// TwinCAT 3 PLC project DL_Cryo
// ProgramVersion: 3.1.4023.0
// libraries:
//   ESO LDC Comm Common Library, * (ESO)
//   ESO LDC Comm Serial Library, * (ESO)
//   ESO LDC Motor Library, * (ESO)
//   ESO LDC Shutter Library, * (ESO)
//   ESO LDC Timer Library, * (ESO)
//   Tc2_Standard, * (Beckhoff Automation GmbH)
//   Tc2_System, * (Beckhoff Automation GmbH)
//   Tc2_Utilities, * (Beckhoff Automation GmbH)
//   Tc3_Module, * (Beckhoff Automation GmbH)
//   VisuDialogs, * (System)
//   VisuSymbols,3.5.10.0,System
// project tree:
//   / CameraTrigIO.TcTTO, GlobalTextList.TcGTLO, PlcTask.TcTTO
//   DUTs/Enumerator/Devices/ E_JANSSEN_CADM2_FAIL_SAFE_STATE.TcDUT, E_JANSSEN_CMD_TYPE.TcDUT, E_JANSSEN_ERROR.TcDUT, E_JANSSEN_STATUS.TcDUT, E_SA_CH_CMD.TcDUT, E_SA_CH_ERROR.TcDUT, E_SA_POS_ELT_STATE.TcDUT, E_SA_POS_ELT_SUBSTATE.TcDUT, E_SA_POS_SM_STATE.TcDUT, E_SA_RPC_ERROR.TcDUT
//   DUTs/Structures/Comm/ T_JANSSEN_CALIBTATION_VALUES.TcDUT
//   DUTs/Structures/Devices/ T_JANSSEN_CFG.TcDUT, T_JANSSEN_CH_CTRL.TcDUT, T_JANSSEN_COMMAND.TcDUT, T_JANSSEN_CTRL.TcDUT, T_JANSSEN_INFO.TcDUT, T_JANSSEN_READING.TcDUT, T_JANSSEN_STAT.TcDUT, T_SA_CH_STATE.TcDUT, T_SA_DEV_STATUS.TcDUT, T_SCIFY_FILTER_WHEEL_CFG.TcDUT, T_SCIFY_FILTER_WHEEL_STAT.TcDUT
//   GVLs/ GVL_Cryo_Temperatures.TcGVL, GVL_DL_Scanning_Homming.TcGVL
//   POUs/ CameraTrig.TcPOU, FB_Cryostat_State.TcPOU, MAIN.TcPOU
//   POUs/FILTER_WHEEL/ FB_SCIFY_FILTER_WHEEL_FW102C.TcPOU
//   VISUs/ DL_Servo_1_Config.TcVIS, DL_Servo_1_Control.TcVIS, Filter_Wheel.TcVIS, GUI_DL_2.TcVIS, GUI_TIME_INFORMATION.TcVIS, Shutter_1.TcVIS, TipTilt_Servo_1.TcVIS, VisualizationManager.TcVMO (not stored)

CONFIGURATION DL_Cryo
    RESOURCE PLC ON TwinCAT3
        TASK CameraTrigIO(INTERVAL := T#1ms, PRIORITY := 1);
        TASK PlcTask(INTERVAL := T#10ms, PRIORITY := 9);
        PROGRAM CameraTrig WITH CameraTrigIO : CameraTrig;
        PROGRAM MAIN WITH PlcTask : MAIN;
    END_RESOURCE
END_CONFIGURATION

// ---- DUTs/Enumerator/Devices/E_JANSSEN_CADM2_FAIL_SAFE_STATE.TcDUT
{attribute 'qualified_only'}
// 'strict' cannot be used since we mix our own codes with TC codes
//{attribute 'strict'}
TYPE E_JANSSEN_CADM2_FAIL_SAFE_STATE :
(
	OK		 						:= 0,
	UPPER_VOLTAGE_RAIL_IS_MISSING,
	LOWER_VOLTAGE_RAIL_IS_MISSING,	
	THERMAL_OVERLOAD,
	OVER_CURRENT_100US_UPPER_RAIL,
	OVER_CURRENT_1MS_UPPER_RAIL,
	OVER_CURRENT_100US_LOWER_RAIL,
	OVER_CURRENT_1MS_LOWER_RAIL	
);
END_TYPE

// ---- DUTs/Enumerator/Devices/E_JANSSEN_CMD_TYPE.TcDUT
{attribute 'qualified_only'}
{attribute 'strict'}
TYPE E_JANSSEN_CMD_TYPE :
(
	INIT := 0,	// Commands for system initialisation
	READ,		// Commands for Reading status
	CFG,		// Commands for Configuring channels
	CTRL		// Commands for Controlling positioners, e.g. CAL, REF, MOVE, STOP
);
END_TYPE

// ---- DUTs/Enumerator/Devices/E_JANSSEN_ERROR.TcDUT
{attribute 'qualified_only'}
{attribute 'strict'}
TYPE E_JANSSEN_ERROR :
(
	OK				:= 16#0000,
	NOT_IN_OP_STATE	:= 16#0001,
	NOT_INIT		:= 16#0002,
	TIMEOUT			:= 16#0004,
	COMM			:= 16#0008,
	WRONG_STATE		:= 16#0010,
	NOT_IDLE		:= 16#0020
);
END_TYPE

// ---- DUTs/Enumerator/Devices/E_JANSSEN_STATUS.TcDUT
{attribute 'qualified_only'}
{attribute 'strict'}
TYPE E_JANSSEN_STATUS :
(
	NOT_INIT	:= -1,
	IDLE		:= 0,
	ERROR		:= 1,
	BUSY		:= 2
);
END_TYPE

// ---- DUTs/Enumerator/Devices/E_SA_CH_CMD.TcDUT
{attribute 'qualified_only'}
{attribute 'strict'}
TYPE E_SA_CH_CMD :
(
	NONE	:= 0,
	RESET,
	CALIB,
	REF,
	ENABLE,
	DISABLE,
	ENABLE_BASE_DRIVE,
	DISABLE_BASE_DRIVE,
	ENABLE_SERVO_DRIVE,
	DISABLE_SERVO_DRIVE,
	ENABLE_FLEX_DRIVE,
	DISABLE_FLEX_DRIVE,
	STOP,
	MOV,
	MOVE_TO_SETPOINT,
	EMERGENCY_STOP,
	SET_POINT_ACHIEVED
);
END_TYPE

// ---- DUTs/Enumerator/Devices/E_SA_CH_ERROR.TcDUT
{attribute 'qualified_only'}
// 'strict' cannot be used since we mix our own codes with TC codes
//{attribute 'strict'}
TYPE E_SA_CH_ERROR :
(
	OK				:= 0,
	HW_NOT_OP,
	CONFIG,				// Configuration problem, e.g. pointers not set.		
	LOCAL,			
	SETPOS,
	STOP,
	
	ABORT,
	SW_LIMIT_LOWER,
	SW_LIMIT_UPPER,
	ENABLE,
	CTRL,				// MCS2 controller error
	COMM				// MCS2 controller communication problem

);
END_TYPE

// ---- DUTs/Enumerator/Devices/E_SA_POS_ELT_STATE.TcDUT
{attribute 'qualified_only'}
{attribute 'strict'}
TYPE E_SA_POS_ELT_STATE :
(
	NONE	:= 0,
	NOTOP,
	OP
);
END_TYPE

// ---- DUTs/Enumerator/Devices/E_SA_POS_ELT_SUBSTATE.TcDUT
{attribute 'qualified_only'}
{attribute 'strict'}
TYPE E_SA_POS_ELT_SUBSTATE :
(
	NONE					:= 0,
	
	NOTOP_NOTREADY			:= 100,
	NOTOP_READY				:= 101,
	NOTOP_INITIALIZING		:= 102,
	NOTOP_ABORTING			:= 107,
	
	NOTOP_ERROR				:= 199,
	
	
	OP_STANDSTILL			:= 216,            
	OP_MOVING				:= 217,
	OP_SETTING_POS			:= 218,
	OP_STOPPING				:= 219,
	
	OP_ERROR				:= 299
);
END_TYPE

// ---- DUTs/Enumerator/Devices/E_SA_POS_SM_STATE.TcDUT
{attribute 'qualified_only'}
{attribute 'strict'}
TYPE E_SA_POS_SM_STATE :
(
	// Positioner State Machine States
	NOT_READY := 0,	// The system just started.
	CALIB,			// The Positioner is Calibrating
	INIT,			// The Positioner is INITialising/REFerencing
	POST_INIT,		// In POST_INIT we calibrate REF and read CFG once.
	CALIB_REF,		// Calibrate REF position.
	READY,			// NOT OPERATIONAL / READY (i.e. REFerenced)
	
	OP,				// Positioner is Operational
	ERROR,			// Positioner is in error
	
	BASE_DRIVE_MODE, // Janssen controller Basic Drive Mode 
	MOVING,			// Positioner is moving in Basic Drive Mode
	
	STOP,			// Positioner is stopping in Basic Drive Mode OR Exiting a Mode
 	
	
	FLEX_DRIVE_MODE, // Janssen controller external input mode
	
	SERVO_DRIVE_MODE, // ENABLE Janssen controller Servo Drive Mode
	DISABLE_SERVO_DRIVE_MODE, //Disable Janssen controller Servo Drive Mode
	MOVING_TO_SETPOINT,// 3 positioners are Moving to their respective set points in Servo Drive Mode
	EMERGENCY_STOP,    // Emergency stop to halt the positioners
	MOVING_TO_SET_POINT 
	
);
END_TYPE

// ---- DUTs/Enumerator/Devices/E_SA_RPC_ERROR.TcDUT
{attribute 'qualified_only'}
//{attribute 'strict'}
TYPE E_SA_RPC_ERROR :
(
	OK						:= 0,
	NOT_OP					:= -1,			
	NOT_NOTOP_READY			:= -2,			
	NOT_NOTOP_NOTREADY		:= -3,			
	LOCAL					:= -4,			
	SW_LIMIT_LOWER			:= -5,			
	SW_LIMIT_UPPER			:= -6,			
	CHANNEL					:= -7,			
	VEL_ZERO				:= -8,			
	VEL_NEG					:= -9,			
	VEL_MAX					:= -10,			
	CH_NOT_OP				:= -11,
	CTRL_ERROR				:= -12,
	MOVING					:= -13,
	COMM					:= -14	// MCS2 Controller communication problem			
);
END_TYPE

// ---- DUTs/Structures/Comm/T_JANSSEN_CALIBTATION_VALUES.TcDUT
TYPE T_JANSSEN_CALIBTATION_VALUES :
STRUCT
	nGainSetting:				DINT;
	nUpperThresholdValue:		DINT;
	nLowerThresholdValue:		DINT;
END_STRUCT
END_TYPE

// ---- DUTs/Structures/Devices/T_JANSSEN_CFG.TcDUT
TYPE T_JANSSEN_CFG EXTENDS T_RS_BASE_CFG :
STRUCT
	
    //
	// List of Monitoring commands in PRE-OPERATION.
	// Executed before the Positioner has been Referenced/initialised.
	//
	{attribute 'OPC.UA.DA' := '0'}
	cmdList_NOT_READY:	ARRAY [0..15] OF T_JANSSEN_COMMAND := [
							(cmd := 'GFS 1',     	nReplies := 1),
							(cmd := 'GFS 2',     	nReplies := 1),
							(cmd := 'GFS 3',     	nReplies := 1),
							(cmd := 'FBXT', 		nReplies := 1),
							(cmd := 'STP 1', 		nReplies := 1),
							(cmd := 'STP 2', 		nReplies := 1),
							(cmd := 'STP 3', 		nReplies := 1),
							(cmd := '', 			nReplies := 0),
							(cmd := '', 			nReplies := 0)];
	//
	// INIT commands.
	// Executed during Initialisation, before going to OPERATIONAL.
	//
	{attribute 'OPC.UA.DA' := '0'}
	cmdList_Init:	ARRAY [0..7] OF T_JANSSEN_COMMAND := [							
							(cmd := '/GBR USB', 	nReplies := 1),
							(cmd := '', 			nReplies := 0)];

	//
	// List of commands to SET Channel/Positioner Configuration.
	// Note the # and *** characters !!!
	// The actual command will be set like this:
	//    #   will be replaced with channel number
	//    *** will be replaced with a value
	// Example:
	//    ':CHAN#:PCON:OPT ***' => ':CHAN1:PCON:OPT 256'
	//
	// Important NOTE:
	// At this stage RLIM:MIN and RLIM:MAX are disabled, i.e. = 0.
	// The actual limits will be set at the E_SA_POS_SM_STATE.CALIB_REF stage,
	// see M_SetCmdList().
	//
	// These commands are sent only once, just before the positioner is 
	// commanded to Reference (INIT).
	//
	{attribute 'OPC.UA.DA' := '0'}
	cmdList_CfgSet:	ARRAY [0..15] OF T_JANSSEN_COMMAND := [						
							(cmd := '/GBR RS422', 			nReplies := 1),
							(cmd := '/MODLIST', 			nReplies := 1),
							(cmd := 'FBXT', 				nReplies := 1),
							(cmd := 'STP 1', 				nReplies := 1),
							(cmd := 'STP 2', 				nReplies := 1),
							(cmd := 'STP 3', 				nReplies := 1),
							(cmd := 'MLS 4 1', 				nReplies := 1), // Get calibration values
							(cmd := 'MLS 4 2', 				nReplies := 1), // Get calibration values
							(cmd := 'MLS 4 3', 				nReplies := 1), // Get calibration values
							(cmd := 'FBST', 				nReplies := 1), //// Get status position control
							//(cmd := '/VER', 		nReplies := 1),
							//(cmd := 'FBEN CBS10-RLS 300 CBS10-RLS 300 CBS10-RLS 300 1 293', 	nReplies := 1),
							(cmd := '', 					nReplies := 0),			
							//(cmd := ':CHAN#:INP:THR ***', 		nReplies := 0),							
							//(cmd := ':CHAN#:RLIM:MIN 0', 		nReplies := 0),
							(cmd := '', 		nReplies := 0)];
							

	//				
	// List of commands to GET Channel/Positioner Configuration.
	// These commands are sent from the moment the SW started till the positioner 
	// has been Calibrated or Referenced (INIT).
	// Once the Positioer is Ready, these commans are not sent any more.
	//
	{attribute 'OPC.UA.DA' := '0'}
	cmdList_POST_INIT:	ARRAY [0..15] OF T_JANSSEN_COMMAND := [							
							(cmd := '/VER', 		nReplies := 1),
							(cmd := '', 		nReplies := 0)];
							

	

	//
	// List of Monitoring commands in OPERATION.
	// Executed once the Positioner has been Referenced/initialised.
	//
	{attribute 'OPC.UA.DA' := '0'}
	cmdList_Mon:	ARRAY [0..15] OF T_JANSSEN_COMMAND := [
							(cmd := 'GFS 1', 	nReplies := 1),
							(cmd := 'GFS 2', 	nReplies := 1),
							(cmd := 'GFS 3', 	nReplies := 1),
							(cmd := 'FBST', 	nReplies := 1),
							(cmd := 'CGVA 4', 	nReplies := 1),						
							(cmd := '', 		nReplies := 0)];
							
	// Janssen controller flex drive mode
	//Command EXT [ADDR] [DIR] [FREQ] [RSS] [TEMP] [STAGE] [DF]
	cmdList_enable_flex_drive:		ARRAY [0..15] OF T_JANSSEN_COMMAND := [
										(cmd := 'EXT 1 1 600 100 293 CLA2601 1', 	nReplies := 1),						
										(cmd := '', 		nReplies := 0)];
	//Disable flex drive
	//Command FBXT
	//Response (example) Control loop disabled.
	cmdList_disable_flex_drive:	ARRAY [0..15] OF T_JANSSEN_COMMAND := [
										(cmd := 'STP 1', 	nReplies := 1),
										(cmd := 'STP 2', 	nReplies := 1),
										(cmd := 'STP 3', 	nReplies := 1),						
										(cmd := '', 		nReplies := 0)];

	// Janssen controller Servo Drive Mode
	// Command FBEN [STAGE1] [FREQ1] [STAGE2] [FREQ2] [STAGE3] [FREQ3] [DF] [TEMP]		
	cmdList_enable_servo_drive:	ARRAY [0..15] OF T_JANSSEN_COMMAND := [
								(cmd := 'FBEN CBS10-RLS 300 CBS10-RLS 300 CBS10-RLS 300 1 293', 	nReplies := 1),						
								(cmd := '', 		nReplies := 0)];
								
	//Disable servo drive
	//Command FBXT
	//Response (example) Control loop disabled.
	cmdList_disable_servo_drive:	ARRAY [0..15] OF T_JANSSEN_COMMAND := [
								(cmd := 'FBXT', 	nReplies := 1),
								(cmd := 'STP 1', 	nReplies := 1),
								(cmd := 'STP 2', 	nReplies := 1),
								(cmd := 'STP 3', 	nReplies := 1),						
								(cmd := '', 		nReplies := 0)];
	
	// 3 positioners are Moving to their respective set points in Servo Drive Mode
	//Command FBCS [SP1] [ABS] [SP2] [ABS] [SP3] [ABS]
	//Command (example, SP in [m]) FBCS -1e-3 0 1e-3 1 1.23e-4 1
	//Command (example, SP in [rad]) FBCS 6.28 0 0 0 0 0
	//Response (example) Control loop setpoints set.
	
	cmdList_moving_to_setpoint:	ARRAY [0..15] OF T_JANSSEN_COMMAND := [
								(cmd := 'FBCS -1e-3 0 1e-3 1 1.23e-4 1', 	nReplies := 1),						
								(cmd := '', 		nReplies := 0)];
								
	// Emergency stop to halt the positioners
	cmdList_emergency_stop: ARRAY [0..15] OF T_JANSSEN_COMMAND := [
								(cmd := 'FBES', 	nReplies := 1),						
								(cmd := '', 		nReplies := 0)];
								
	// CSZ – Reset current counter value to zero
	//Command CSZ [ADDR] [CH]
	//Command (example) CSZ 4 1
	//Response (example) Position counter set to 0.
	cmdList_reset_counter_to_zero: ARRAY [0..15] OF T_JANSSEN_COMMAND := [
								(cmd := 'CSZ 4 1', 	nReplies := 1),						
								(cmd := '', 		nReplies := 0)];

	//
	// Array of used channels. Set to TRUE for each used channel.
	// 18 channels max. 6 modules [0..5], 3 connections each [CH1, CH2, CH3].
	// channel = (Module x 3) + (CH-1)
	// For example:
	//   First connection (CH1) of first module (Module0): channel = 0 x 3 + (1-1) = 0
	//   Second connection (CH2) of first module (Module0): channel = 0 x 3 + (2-1) = 1
	//   Third connection (CH3) of third module (Module2): channel = 2 x 3 + (3-1) = 8
	//  
	arrUsedCh:	ARRAY [0..17] 	OF BOOL;	

	//
	// Array of used modules. Set to TRUE for each used module.
	// Automatically populated in method M_Configure().
	//
	arrUsedMod:	ARRAY [0..5] 	OF BOOL;	
	
	// Channel configuration structures
//	arrChCfg:	ARRAY [0..17] OF T_SA_CH_CFG;		

(*
	JANSSEN_GET_BR:		STRING(10) := '/GBR RS422';
	JANSSEN_GET_VER:	STRING(8) := '/VER';
	JANSSEN_MODLIST:	STRING(8) := '/MODLIST';
	//CCC_CMD_GET_VERS:	STRING(8) := '>00V??';
	CCC_CMD_GET_VERS:	STRING(8) := '/GBR';
	//CCC_CMD_RESET:		STRING(8) := '>00u??';
	CCC_CMD_RESET:		STRING(8) := '/GBR';
	CCC_CMD_GET_TEMP:	STRING(8) := '>00H??';
	CCC_CMD_GET_FLOW:	STRING(8) := '>00f??';
	//CCC_CMD_GET_STAT:	STRING(8) := '>00o??';
	CCC_CMD_GET_STAT:	STRING(8) := '/GBR';
	CCC_CMD_SET_HOST:	STRING(8) := '>00J??';
	CCC_CMD_SET_THST:	STRING(8) := '>00T??';
	CCC_CMD_SET_TAMB:	STRING(8) := '>00t??';

	(* List of INIT commands *)
	cmdList_Init:	ARRAY [1..4] OF T_JANSSEN_COMMAND := [
							//(cmd := CCC_CMD_RESET, 		nValues := 4),
							//(cmd := CCC_CMD_GET_VERS, 	nValues := 4),
							//(cmd := CCC_CMD_RESET, 		nValues := 0),
							//(cmd := CCC_CMD_GET_VERS, 	nValues := 0),
							//(cmd := JANSSEN_GET_BR, 	nValues := 4),
							//(cmd := '', 				nValues := 0),
							(cmd := '', 				nValues := 0),
							(cmd := '', 				nValues := 0),
							(cmd := '', 				nValues := 0),
							(cmd := '', 				nValues := 0)];


	(*	List of READ commands *)
	cmdList_Read:	ARRAY [1..4] OF T_JANSSEN_COMMAND := [
							//(cmd := CCC_CMD_GET_STAT, 	nValues := 5), (* 5 bytes *)
							//(cmd := CCC_CMD_GET_TEMP, 	nValues := 5), (* 5 words = 10 bytes*)
							//(cmd := CCC_CMD_GET_FLOW, 	nValues := 3), (* 3 words = 6 bytes *)
							//(cmd := JANSSEN_GET_BR, 	nValues := 4),
							(cmd := '/GBR RS422',       nValues := 1),
							(cmd := '/GBR USB', 		nValues := 1),
							(cmd := '', 				nValues := 0),
							(cmd := '', 				nValues := 0)];
		*)
					

END_STRUCT
END_TYPE

// ---- DUTs/Structures/Devices/T_JANSSEN_CH_CTRL.TcDUT
TYPE T_JANSSEN_CH_CTRL :
STRUCT
	//
	// Control structure for a single channel/positioner.
	//
	
	//
	// Active command.
	// Setting nCmd to something other than NONE will
	// trigger execution of commands REF, STOP, MOV.
	//
	nCmd:	E_SA_CH_CMD := E_SA_CH_CMD.NONE;	// Active command
	
	
	// JANSSEN Servo Drive Mode. METIS CFO PSM
	
	// Enable Servodrive
	
	sStage1:	STRING	:= 'CBS10-RLS'; // Mention here the correct stage
	sStage2:	STRING	:= 'CBS10-RLS'; // Mention here the correct stage
	sStage3:	STRING	:= 'CBS10-RLS'; // Mention here the correct stage
	
	// Step Frequency [1 to 600]
	
	nFreq1:		DINT	:= 300; // Step frequency for actuator 1
	nFreq2:		DINT	:= 300; // Step frequency for actuator 2
	nFreq3:		DINT	:= 300; // Step frequency for actuator 3
	
	// Operating Temperturte
	
	nTemp:		DINT; // In Kelvin
	
	// Drive Factor: 
	
	lrDriveFactor:	LREAL := 1.0; // [0.1 to 3.0] In normal operating conditions, set this value to 1 (or 1.0).
	
	// Setpoints
	lrSetPoint1 : LREAL; //Setpoint 1 position in [m]
	lrSetPoint2 : LREAL; //Setpoint 1 position in [m]
	lrSetPoint3 : LREAL; //Setpoint 1 position in [m]
	
	// Set [ABS] to 1 to enable absolute positioning, otherwise set to 0 (zero). 
	// When using COE / OEM2: absolute positioning is relative to count 0 (zero)9 , 
	//whereas relative positioning is relative to the current count value.
	
	bAbsolutePositioning1 : BOOL;
	bAbsolutePositioning2 : BOOL;
	bAbsolutePositioning3 : BOOL;
	
	//SA
	lrPos:	LREAL;		// Position in User Units, i.e. [deg] or [mm]
	lrOff:	LREAL;		// Position offset in User Units, i.e. [deg] or [mm]
	lrVel:	LREAL;		// Velocity in User Units, i.e. [deg/s] or [mm/sec]
	
END_STRUCT
END_TYPE

// ---- DUTs/Structures/Devices/T_JANSSEN_COMMAND.TcDUT
TYPE T_JANSSEN_COMMAND :
STRUCT
	cmd:		STRING := '';	(* Command to send *)
	nReplies:	UINT;   		(* Number of replies, i.e. reply terminators *)
END_STRUCT
END_TYPE

// ---- DUTs/Structures/Devices/T_JANSSEN_CTRL.TcDUT
TYPE T_JANSSEN_CTRL EXTENDS T_RS_BASE_CTRL :
STRUCT
	// Arrays of structures for Configuration and Control commands.
	// Note that only one positioner is handled in each monitoring cycle.
	{attribute 'OPC.UA.DA' := '0'}
	cmdList:			ARRAY [0..15]	OF T_JANSSEN_COMMAND;	// List of up to 16 Commands per channel
	
END_STRUCT
END_TYPE

// ---- DUTs/Structures/Devices/T_JANSSEN_INFO.TcDUT
TYPE T_JANSSEN_INFO :
STRUCT
(*
	Driver Information

	Change LOG:
	1.0	12/02/2014	- Ported from TC2.
	1.1	13/02/2014	- Addition of input parameters for Model and readout period.
	1.2	20/02/2014	- E_CCC_STATUS.ERROR := 1, to match IODev ICD.
					- Disabled OPC UA for comm instance of FB_RS_COMM.
					- Fixed bug in INIT (wrong pointer used)
					- Bytes swapped for Temperatures and Flows.
					- On error, all values set to 9999. Alarm activated.
	1.3 07/11/2014	- Newest version always for References.
					- Remove Tc2_OpcUa library from References.
					- Renamed library to CCC.library (was CCC_TC3.library)
					- Created lib directory.
	1.4 10/02/2016	- On reboot, the device is in NOT INIT (no error!)
					- On INIT start, error is cleared.
	2.0 2016-08-10	- OPC UA notation with TMC Files
	2.1 2017-02-03	- sCmdSuffix and sReplySuffix passed to comm instance.

*)
	sDate:			STRING(16)	:= '2017-02-03';
	sDescription:	STRING(32) 	:= 'Cabinet Cooling Controller';
	sName:			STRING(16)	:= 'FB_CCC';
	sPlatform:		STRING(16)	:= 'CoDeSys';
	sSynopsis:		STRING(48)	:= 'Cabinet Cooling Controller for models 1HE & 4HE';
	nVersionMajor:	DINT		:= 2;
	nVersionMinor:	DINT		:= 1;

END_STRUCT
END_TYPE

// ---- DUTs/Structures/Devices/T_JANSSEN_READING.TcDUT
TYPE T_JANSSEN_READING :
STRUCT
	Value:	LREAL;
END_STRUCT
END_TYPE

// ---- DUTs/Structures/Devices/T_JANSSEN_STAT.TcDUT
TYPE T_JANSSEN_STAT EXTENDS T_RS_BASE_STAT :
STRUCT
	(* STAT *)
	nRetries:			INT := 0;			// Total number of retries in case of communication problems
	
	bPeriodic:			BOOL := FALSE;		(* Flag if device is reading periodically *)

	sReply:				STRING; 			(* Last Reply to predefined commands*)
	
	sRandomtext_1:				STRING;
	sRandomtext_2:				STRING;
	sRandomtext_3:				STRING;
	sRandomtext_4:				STRING;
	sRandomtext_5:				STRING;
	sRandomtext_6:				STRING;
	sRandomtext_7:				STRING;
	sRandomtext_8:				STRING;
	
	sDeviceID:			STRING(48);
	
	(*Baut rate *)
	sBaud_rate_RS422: 			STRING;
	sBaud_rate_USB: 			STRING;
	sFirmware_Version:			STRING;
	sChannel_1_Stop:			STRING;
	sChannel_2_Stop:			STRING;
	sChannel_3_Stop:			STRING;
	
	sFailSafeState_1:			STRING;
	sFailSafeState_2:			STRING;
	sFailSafeState_3:			STRING;
	
	//  
			
	
	// FBST – Get status position control
	sPositionControlStatus:		STRING;
	
	bPositionControl:			BOOL;
	bMovingToSetPoint:			BOOL;
	bInvalidSetPoint_1:			BOOL;
	bInvalidSetPoint_2:			BOOL;
	bInvalidSetPoint_3:			BOOL;
	
	
	nPositionError_1:			DINT;
	nPositionError_2:			DINT;
	nPositionError_3:			DINT;
	
	// MLS Get calibration values
	sCalibrationValues:			STRING;
	
	nCalibrationValues_Cannel_1:	T_JANSSEN_CALIBTATION_VALUES;
	nCalibrationValues_Cannel_2:	T_JANSSEN_CALIBTATION_VALUES;
	nCalibrationValues_Cannel_3:	T_JANSSEN_CALIBTATION_VALUES;
	
	// CGVA 4 counter values of all three channels
	sCounterValues:				STRING;
	
	nCounterValue_Channel_1:		DINT;
	nCounterValue_Channel_2:		DINT;
	nCounterValue_Channel_3:		DINT;
	
	// Command Error
	sCommandError:				STRING;
	
	//Emergency Stop
	bEmergencyStopEnabled:		BOOL;
	
	//FBCS – Go to setpoint -> Control loop setpoints set
	bPositionControlLoop:		BOOL;
	
	//Servo Drive Control
	bServoDrive:				BOOL:= FALSE;
	sServoDriveStatus:			STRING;
	
	//Flex Control
	bFlexDrive:					BOOL;
	
	// /MODLIST Get a list of all installed modules
	
	sInstalledModules:			ARRAY[1..6] OF STRING;
	
	// CGVA – Get current counter value of all channels
	
	nCounterValues:				ARRAY[1..3] OF DINT;
	
	// Get calibration values.  command specific for Basedrive mode of operation
	//Command MLS [ADDR] [CH]
	//Response [GAIN],[UT],[LT]
	
	sCalibValues_1:				STRING;
	sCalibValues_2:				STRING;
	sCalibValues_3:				STRING;

		
	
	
	
	
	(* Status retrieved with command CCC_CMD_GET_STAT *)
	(* decode CSTAT1 byte *)
	bWarn_cabinet_high:			BOOL;
	bWarn_cabinet_no_control:	BOOL;
	bWarn_outlet_high:			BOOL;
	bWarn_inlet_high:			BOOL;
	bWarn_airflow_insufficient:	BOOL;
	bWarn_coolant_insufficient:	BOOL;
	bWarn_door_open:			BOOL;
	bWarn_relay1_warning:		BOOL;
	bWarn_relay2_alarm:			BOOL;

	(* decode CSTAT2 byte *)
	bFault_temp_sensor_ambient:	BOOL;
	bFault_temp_sensor_cabinet:	BOOL;
	bFault_temp_sensor_inlet:	BOOL;
	bFault_temp_sensor_outlet:	BOOL;
	bFault_analog_supply:		BOOL;
	bFault_digital_supply:		BOOL;
	
	(* Temperatures [degC] retrieved with command CCC_CMD_GET_TEMP *)
	lrTemp_outlet:	LREAL;
	lrTemp_inlet:	LREAL;
	lrTemp_cabinet:	LREAL;
	lrTemp_ambient:	LREAL;
	
	(* Flows [l/h] retrieved with command CCC_CMD_GET_FLOW *)
	lrFlow_1:		LREAL;
	lrFlow_2:		LREAL;
	lrFlow_3:		LREAL;
	
	// SmarACT STATs
	
	//bLocal:			BOOL	:= FALSE;	// if TRUE, device operated from PLC GUI 

	//nErrorCode: 	E_SA_CH_ERROR 	:= E_SA_CH_ERROR.OK;	// Error code 
	//nRpcErrorCode: 	E_SA_RPC_ERROR 	:= E_SA_RPC_ERROR.OK;	// RPC Error code

	bCtrlCommProblem:	BOOL;			// SmarAct MCS2 Controller Comm Problem
	//nCtrlErrorCode: E_SM_ERROR;			// SmarAct MCS2 Controller Error code
	nCtrlState:		E_RS_BASE_STATE;	// SmarAct MCS2 Controller State	

	//sErrorText: 	STRING 	:= 'OK'; 			// Error text 
	//sRpcErrorText: 	STRING 	:= 'OK'; 			// RPC Error text 
	//sStatus: 		STRING 	:= 'OK'; 			// Status in textual form, e.g. 'OFF' 
	
	//
	// Standard ELT States and Substates
	//
	//nState:			E_SA_POS_ELT_STATE 		:= E_SA_POS_ELT_STATE.NOTOP;
	//nSubstate:		E_SA_POS_ELT_SUBSTATE	:= E_SA_POS_ELT_SUBSTATE.NOTOP_NOTREADY;
	
	//sState:			STRING	:= 'NOTOP';
	//sSubstate:		STRING	:= 'NOT READY';

	//
	// Positioner State Machine State.
	// Depending on the State, different command sets will be executed.
	//
	nPosState:			E_SA_POS_SM_STATE := E_SA_POS_SM_STATE.NOT_READY;
	nLastPosState:		E_SA_POS_SM_STATE := E_SA_POS_SM_STATE.NOT_READY;
	

	lrPosTarget:		LREAL;			// Target  position in User Units
	lrPosActual:		LREAL;			// Current position in User Units

	//bConfigured:		BOOL;			// Flag if M_Configure has been executed.	
	bError:				BOOL;
	bEnabled:			BOOL;			// Flag if axis is enabled
	//bInitialised:		BOOL;			// Flag if positioner has been initialised/referenced
	bInPosition:		BOOL;			// Flag if axis is In-Position

	//
	// Channel State parameters read from the controller
	// A channel is a Positioner.
	//
	nCH_STATE:				UDINT;			// Positioner State as UDINT
	{attribute 'OPC.UA.DA' := '0'}
	stState:			T_SA_CH_STATE;	// Positioner State structure, from nSTATE
	
	//
	// Device/Channel/Positioner status in user units, i.e. [pm] and [nd].
	// These values are read periodically.
	// Values are normally huge, e.g. pos=18000000000 [nd].
	//
	{attribute 'OPC.UA.DA' := '0'}
	devStatus:			T_SA_DEV_STATUS; 

END_STRUCT
END_TYPE

// ---- DUTs/Structures/Devices/T_SA_CH_STATE.TcDUT
TYPE T_SA_CH_STATE :
STRUCT
	//
	// Channel State
	// Got with the ':CHAN#:STAT?' command
	//
	bBASE_DRIVE_ENABLED:			BOOL;
	bFLEX_DRIVE_ENABLED:			BOOL;
	bSERVO_DRIVE_ENABLED:			BOOL;
	
	bACTIVELY_MOVING:			BOOL;
	bCLOSED_LOOP_ACTIVE:		BOOL;
	bCALIBRATING:				BOOL;
	bREFERENCING:				BOOL;
	bMOVE_DELAYED:				BOOL;
	bSENSOR_PRESENT:			BOOL;
	bIS_CALIBRATED:				BOOL;
	bIS_REFERENCED:				BOOL;
	bEND_STOP_REACHED:			BOOL;
	bRANGE_LIMIT_REACHED:		BOOL;
	bFOLLOWING_LIMIT_REACHED:	BOOL;
	bMOVEMENT_FAILED:			BOOL;
	bIS_STREAMING:				BOOL;
	bPOSITIONER_OVERLOAD:		BOOL;
	
	bOVER_TEMPERATURE:			BOOL;
	
	bREFERENCE_MARK:			BOOL;
	bIS_PHASED:					BOOL;
	bPOSITIONER_FAULT:			BOOL;
	bAMPLIFIER_ENABLED:			BOOL;
	bIN_POSITION:				BOOL;

	bERROR:						BOOL := TRUE;
	bControllerStateError:			BOOL := TRUE;
END_STRUCT
END_TYPE

// ---- DUTs/Structures/Devices/T_SA_DEV_STATUS.TcDUT
//
// Device/Channel/Positioner status in user units, i.e. [pm] and [nd]
//
TYPE T_SA_DEV_STATUS :
STRUCT
	nCAL_OPT:			DINT;			// Calibration option
	nREF_OPT:			DINT;			// Referencing option
	nPCON_OPT:			DINT;			// Positioner Control Options, 256-'in-pos' flag
	nCLIN:				DINT;			// Control Loop Input, 1-SENSOR
	nTUN_BASE_UNIT:		DINT;			// Positioner Base Unit, 2-meter, 3-degree
	nTUN_BASE_RES:		DINT;			// Positioner Base Resolution, 1x10-9 or 1x10-12
	nTUN_MTYP:			DINT;			// Positioner Movement Type, 0-linear, 1-rotation, etc
	nTUN_RTYP:			DINT;			// Positioner Reference Type, 2-SINGLE_CODED
	nINP_THR:			DINT;			// In Position Threshold [DevU]
	nINP_DEL:			DINT;			// In Position Delay [ms]
	nRLIM_MIN:			LINT;			// MIN Limit [DevU]
	nRLIM_MAX:			LINT;			// MAX Limit [DevU]

	lnPosTarget:		LINT;			// Target  position in Positioner Units
	lnPosActual:		LINT;			// Current position in Positioner Units

END_STRUCT
END_TYPE

// ---- DUTs/Structures/Devices/T_SCIFY_FILTER_WHEEL_CFG.TcDUT
TYPE T_SCIFY_FILTER_WHEEL_CFG EXTENDS T_RS_BASE_CFG :
STRUCT
	
    //
	// List of Monitoring commands in PRE-OPERATION.
	// Executed before the Positioner has been Referenced/initialised.
	//
	{attribute 'OPC.UA.DA' := '0'}
	cmdList_NOT_READY:	ARRAY [0..15] OF T_JANSSEN_COMMAND := [
							(cmd := '*idn?',     	nReplies := 1),
							(cmd := 'pos?',     	nReplies := 1),
							(cmd := 'speed?',     	nReplies := 1),
							(cmd := 'sensors?', 		nReplies := 1),
							(cmd := 'baud?', 		nReplies := 1),
							(cmd := '', 			nReplies := 0),
							(cmd := '', 			nReplies := 0)];
	//
	// INIT commands.
	// Executed during Initialisation, before going to OPERATIONAL.
	//
	{attribute 'OPC.UA.DA' := '0'}
	cmdList_Init:	ARRAY [0..7] OF T_JANSSEN_COMMAND := [							
							(cmd := 'pos?',     	nReplies := 1),
							(cmd := '', 			nReplies := 0)];

	//
	// List of commands to SET Channel/Positioner Configuration.
	// Note the # and *** characters !!!
	// The actual command will be set like this:
	//    #   will be replaced with channel number
	//    *** will be replaced with a value
	// Example:
	//    ':CHAN#:PCON:OPT ***' => ':CHAN1:PCON:OPT 256'
	//
	// Important NOTE:
	// At this stage RLIM:MIN and RLIM:MAX are disabled, i.e. = 0.
	// The actual limits will be set at the E_SA_POS_SM_STATE.CALIB_REF stage,
	// see M_SetCmdList().
	//
	// These commands are sent only once, just before the positioner is 
	// commanded to Reference (INIT).
	//
	{attribute 'OPC.UA.DA' := '0'}
	cmdList_CfgSet:	ARRAY [0..15] OF T_JANSSEN_COMMAND := [						
							(cmd := 'pos=5', 	nReplies := 1),
							(cmd := '', 			nReplies := 0)];
							

	//				
	// List of commands to GET Channel/Positioner Configuration.
	// These commands are sent from the moment the SW started till the positioner 
	// has been Calibrated or Referenced (INIT).
	// Once the Positioer is Ready, these commans are not sent any more.
	//
	{attribute 'OPC.UA.DA' := '0'}
	cmdList_POST_INIT:	ARRAY [0..15] OF T_JANSSEN_COMMAND := [							
							(cmd := '/VER', 		nReplies := 1),
							(cmd := '', 		nReplies := 0)];
							

	

	//
	// List of Monitoring commands in OPERATION.
	// Executed once the Positioner has been Referenced/initialised.
	//
	{attribute 'OPC.UA.DA' := '0'}
	cmdList_Mon:	ARRAY [0..15] OF T_JANSSEN_COMMAND := [
							(cmd := '*idn?',     	nReplies := 1),
							(cmd := 'pos?',     	nReplies := 1),
							(cmd := 'speed?',     	nReplies := 1),
							(cmd := 'sensors?', 	nReplies := 1),
							(cmd := 'baud?', 		nReplies := 1),
							(cmd := '', 			nReplies := 0),			
							(cmd := '', 			nReplies := 0)];
							
	// Janssen controller flex drive mode
	//Command EXT [ADDR] [DIR] [FREQ] [RSS] [TEMP] [STAGE] [DF]
	cmdList_enable_flex_drive:		ARRAY [0..15] OF T_JANSSEN_COMMAND := [
										(cmd := 'EXT 1 1 600 100 293 CLA2601 1', 	nReplies := 1),						
										(cmd := '', 		nReplies := 0)];
	//Disable flex drive
	//Command FBXT
	//Response (example) Control loop disabled.
	cmdList_disable_flex_drive:	ARRAY [0..15] OF T_JANSSEN_COMMAND := [
										(cmd := 'STP 1', 	nReplies := 1),
										(cmd := 'STP 2', 	nReplies := 1),
										(cmd := 'STP 3', 	nReplies := 1),						
										(cmd := '', 		nReplies := 0)];

	// Janssen controller Servo Drive Mode
	// Command FBEN [STAGE1] [FREQ1] [STAGE2] [FREQ2] [STAGE3] [FREQ3] [DF] [TEMP]		
	cmdList_enable_servo_drive:	ARRAY [0..15] OF T_JANSSEN_COMMAND := [
								(cmd := 'FBEN CBS10-RLS 300 CBS10-RLS 300 CBS10-RLS 300 1 293', 	nReplies := 1),						
								(cmd := '', 		nReplies := 0)];
								
	//Disable servo drive
	//Command FBXT
	//Response (example) Control loop disabled.
	cmdList_disable_servo_drive:	ARRAY [0..15] OF T_JANSSEN_COMMAND := [
								(cmd := 'FBXT', 	nReplies := 1),
								(cmd := 'STP 1', 	nReplies := 1),
								(cmd := 'STP 2', 	nReplies := 1),
								(cmd := 'STP 3', 	nReplies := 1),						
								(cmd := '', 		nReplies := 0)];
	
	// 3 positioners are Moving to their respective set points in Servo Drive Mode
	//Command FBCS [SP1] [ABS] [SP2] [ABS] [SP3] [ABS]
	//Command (example, SP in [m]) FBCS -1e-3 0 1e-3 1 1.23e-4 1
	//Command (example, SP in [rad]) FBCS 6.28 0 0 0 0 0
	//Response (example) Control loop setpoints set.
	
	cmdList_moving_to_setpoint:	ARRAY [0..15] OF T_JANSSEN_COMMAND := [
								(cmd := 'FBCS -1e-3 0 1e-3 1 1.23e-4 1', 	nReplies := 1),						
								(cmd := '', 		nReplies := 0)];
								
	// Emergency stop to halt the positioners
	cmdList_emergency_stop: ARRAY [0..15] OF T_JANSSEN_COMMAND := [
								(cmd := 'FBES', 	nReplies := 1),						
								(cmd := '', 		nReplies := 0)];
								
	// CSZ – Reset current counter value to zero
	//Command CSZ [ADDR] [CH]
	//Command (example) CSZ 4 1
	//Response (example) Position counter set to 0.
	cmdList_reset_counter_to_zero: ARRAY [0..15] OF T_JANSSEN_COMMAND := [
								(cmd := 'CSZ 4 1', 	nReplies := 1),						
								(cmd := '', 		nReplies := 0)];

	//
	// Array of used channels. Set to TRUE for each used channel.
	// 18 channels max. 6 modules [0..5], 3 connections each [CH1, CH2, CH3].
	// channel = (Module x 3) + (CH-1)
	// For example:
	//   First connection (CH1) of first module (Module0): channel = 0 x 3 + (1-1) = 0
	//   Second connection (CH2) of first module (Module0): channel = 0 x 3 + (2-1) = 1
	//   Third connection (CH3) of third module (Module2): channel = 2 x 3 + (3-1) = 8
	//  
	arrUsedCh:	ARRAY [0..17] 	OF BOOL;	

	//
	// Array of used modules. Set to TRUE for each used module.
	// Automatically populated in method M_Configure().
	//
	arrUsedMod:	ARRAY [0..5] 	OF BOOL;	
	
	// Channel configuration structures
//	arrChCfg:	ARRAY [0..17] OF T_SA_CH_CFG;		

(*
	JANSSEN_GET_BR:		STRING(10) := '/GBR RS422';
	JANSSEN_GET_VER:	STRING(8) := '/VER';
	JANSSEN_MODLIST:	STRING(8) := '/MODLIST';
	//CCC_CMD_GET_VERS:	STRING(8) := '>00V??';
	CCC_CMD_GET_VERS:	STRING(8) := '/GBR';
	//CCC_CMD_RESET:		STRING(8) := '>00u??';
	CCC_CMD_RESET:		STRING(8) := '/GBR';
	CCC_CMD_GET_TEMP:	STRING(8) := '>00H??';
	CCC_CMD_GET_FLOW:	STRING(8) := '>00f??';
	//CCC_CMD_GET_STAT:	STRING(8) := '>00o??';
	CCC_CMD_GET_STAT:	STRING(8) := '/GBR';
	CCC_CMD_SET_HOST:	STRING(8) := '>00J??';
	CCC_CMD_SET_THST:	STRING(8) := '>00T??';
	CCC_CMD_SET_TAMB:	STRING(8) := '>00t??';

	(* List of INIT commands *)
	cmdList_Init:	ARRAY [1..4] OF T_JANSSEN_COMMAND := [
							//(cmd := CCC_CMD_RESET, 		nValues := 4),
							//(cmd := CCC_CMD_GET_VERS, 	nValues := 4),
							//(cmd := CCC_CMD_RESET, 		nValues := 0),
							//(cmd := CCC_CMD_GET_VERS, 	nValues := 0),
							//(cmd := JANSSEN_GET_BR, 	nValues := 4),
							//(cmd := '', 				nValues := 0),
							(cmd := '', 				nValues := 0),
							(cmd := '', 				nValues := 0),
							(cmd := '', 				nValues := 0),
							(cmd := '', 				nValues := 0)];


	(*	List of READ commands *)
	cmdList_Read:	ARRAY [1..4] OF T_JANSSEN_COMMAND := [
							//(cmd := CCC_CMD_GET_STAT, 	nValues := 5), (* 5 bytes *)
							//(cmd := CCC_CMD_GET_TEMP, 	nValues := 5), (* 5 words = 10 bytes*)
							//(cmd := CCC_CMD_GET_FLOW, 	nValues := 3), (* 3 words = 6 bytes *)
							//(cmd := JANSSEN_GET_BR, 	nValues := 4),
							(cmd := '/GBR RS422',       nValues := 1),
							(cmd := '/GBR USB', 		nValues := 1),
							(cmd := '', 				nValues := 0),
							(cmd := '', 				nValues := 0)];
		*)
					

END_STRUCT
END_TYPE

// ---- DUTs/Structures/Devices/T_SCIFY_FILTER_WHEEL_STAT.TcDUT
TYPE T_SCIFY_FILTER_WHEEL_STAT EXTENDS T_RS_BASE_STAT :
STRUCT
	(* STAT *)
	nRetries:			INT := 0;			// Total number of retries in case of communication problems
	
	bPeriodic:			BOOL := FALSE;		(* Flag if device is reading periodically *)

	sReply:				STRING; 			(* Last Reply to predefined commands*)
	
	sRandomtext_1:				STRING;
	sRandomtext_2:				STRING;
	sRandomtext_3:				STRING;
	sRandomtext_4:				STRING;
	sRandomtext_5:				STRING;
	sRandomtext_6:				STRING;
	sRandomtext_7:				STRING;
	sRandomtext_8:				STRING;
	
	
	
	// SCIFY Filter Wheel
	bBaud_rate_RS232: 			BOOL;
	sBaud_rate_RS232: 			STRING;
	
	sDeviceID:					STRING(48);		// Model number and firmware version
	
	sFilterPosition:			STRING;			// Positions 1-6
	nCurrentFilterPosition:			STRING;			
	
	bFilterSensors:				STRING;
	bMoveSpeed:					STRING;
	
	
	
	/////////////
	(*Baut rate *)
	sBaud_rate_RS422: 			STRING;
	sBaud_rate_USB: 			STRING;
	sFirmware_Version:			STRING;
	sChannel_1_Stop:			STRING;
	sChannel_2_Stop:			STRING;
	sChannel_3_Stop:			STRING;
	
	sFailSafeState_1:			STRING;
	sFailSafeState_2:			STRING;
	sFailSafeState_3:			STRING;
	
	//  
			
	
	// FBST – Get status position control
	sPositionControlStatus:		STRING;
	
	bPositionControl:			BOOL;
	bMovingToSetPoint:			BOOL;
	bInvalidSetPoint_1:			BOOL;
	bInvalidSetPoint_2:			BOOL;
	bInvalidSetPoint_3:			BOOL;
	
	
	nPositionError_1:			DINT;
	nPositionError_2:			DINT;
	nPositionError_3:			DINT;
	
	// MLS Get calibration values
	sCalibrationValues:			STRING;
	
	nCalibrationValues_Cannel_1:	T_JANSSEN_CALIBTATION_VALUES;
	nCalibrationValues_Cannel_2:	T_JANSSEN_CALIBTATION_VALUES;
	nCalibrationValues_Cannel_3:	T_JANSSEN_CALIBTATION_VALUES;
	
	// CGVA 4 counter values of all three channels
	sCounterValues:				STRING;
	
	nCounterValue_Channel_1:		DINT;
	nCounterValue_Channel_2:		DINT;
	nCounterValue_Channel_3:		DINT;
	
	// Command Error
	sCommandError:				STRING;
	
	//Emergency Stop
	bEmergencyStopEnabled:		BOOL;
	
	//FBCS – Go to setpoint -> Control loop setpoints set
	bPositionControlLoop:		BOOL;
	
	//Servo Drive Control
	bServoDrive:				BOOL:= FALSE;
	sServoDriveStatus:			STRING;
	
	//Flex Control
	bFlexDrive:					BOOL;
	
	// /MODLIST Get a list of all installed modules
	
	sInstalledModules:			ARRAY[1..6] OF STRING;
	
	// CGVA – Get current counter value of all channels
	
	nCounterValues:				ARRAY[1..3] OF DINT;
	
	// Get calibration values.  command specific for Basedrive mode of operation
	//Command MLS [ADDR] [CH]
	//Response [GAIN],[UT],[LT]
	
	sCalibValues_1:				STRING;
	sCalibValues_2:				STRING;
	sCalibValues_3:				STRING;

		
	
	
	
	
	(* Status retrieved with command CCC_CMD_GET_STAT *)
	(* decode CSTAT1 byte *)
	bWarn_cabinet_high:			BOOL;
	bWarn_cabinet_no_control:	BOOL;
	bWarn_outlet_high:			BOOL;
	bWarn_inlet_high:			BOOL;
	bWarn_airflow_insufficient:	BOOL;
	bWarn_coolant_insufficient:	BOOL;
	bWarn_door_open:			BOOL;
	bWarn_relay1_warning:		BOOL;
	bWarn_relay2_alarm:			BOOL;

	(* decode CSTAT2 byte *)
	bFault_temp_sensor_ambient:	BOOL;
	bFault_temp_sensor_cabinet:	BOOL;
	bFault_temp_sensor_inlet:	BOOL;
	bFault_temp_sensor_outlet:	BOOL;
	bFault_analog_supply:		BOOL;
	bFault_digital_supply:		BOOL;
	
	(* Temperatures [degC] retrieved with command CCC_CMD_GET_TEMP *)
	lrTemp_outlet:	LREAL;
	lrTemp_inlet:	LREAL;
	lrTemp_cabinet:	LREAL;
	lrTemp_ambient:	LREAL;
	
	(* Flows [l/h] retrieved with command CCC_CMD_GET_FLOW *)
	lrFlow_1:		LREAL;
	lrFlow_2:		LREAL;
	lrFlow_3:		LREAL;
	
	// SmarACT STATs
	
	//bLocal:			BOOL	:= FALSE;	// if TRUE, device operated from PLC GUI 

	//nErrorCode: 	E_SA_CH_ERROR 	:= E_SA_CH_ERROR.OK;	// Error code 
	//nRpcErrorCode: 	E_SA_RPC_ERROR 	:= E_SA_RPC_ERROR.OK;	// RPC Error code

	bCtrlCommProblem:	BOOL;			// SmarAct MCS2 Controller Comm Problem
	//nCtrlErrorCode: E_SM_ERROR;			// SmarAct MCS2 Controller Error code
	nCtrlState:		E_RS_BASE_STATE;	// SmarAct MCS2 Controller State	

	//sErrorText: 	STRING 	:= 'OK'; 			// Error text 
	//sRpcErrorText: 	STRING 	:= 'OK'; 			// RPC Error text 
	//sStatus: 		STRING 	:= 'OK'; 			// Status in textual form, e.g. 'OFF' 
	
	//
	// Standard ELT States and Substates
	//
	//nState:			E_SA_POS_ELT_STATE 		:= E_SA_POS_ELT_STATE.NOTOP;
	//nSubstate:		E_SA_POS_ELT_SUBSTATE	:= E_SA_POS_ELT_SUBSTATE.NOTOP_NOTREADY;
	
	//sState:			STRING	:= 'NOTOP';
	//sSubstate:		STRING	:= 'NOT READY';

	//
	// Positioner State Machine State.
	// Depending on the State, different command sets will be executed.
	//
	nPosState:			E_SA_POS_SM_STATE := E_SA_POS_SM_STATE.NOT_READY;
	nLastPosState:		E_SA_POS_SM_STATE := E_SA_POS_SM_STATE.NOT_READY;
	

	lrPosTarget:		LREAL;			// Target  position in User Units
	lrPosActual:		LREAL;			// Current position in User Units

	//bConfigured:		BOOL;			// Flag if M_Configure has been executed.	
	bError:				BOOL;
	bEnabled:			BOOL;			// Flag if axis is enabled
	//bInitialised:		BOOL;			// Flag if positioner has been initialised/referenced
	bInPosition:		BOOL;			// Flag if axis is In-Position

	//
	// Channel State parameters read from the controller
	// A channel is a Positioner.
	//
	nCH_STATE:				UDINT;			// Positioner State as UDINT
	{attribute 'OPC.UA.DA' := '0'}
	stState:			T_SA_CH_STATE;	// Positioner State structure, from nSTATE
	
	//
	// Device/Channel/Positioner status in user units, i.e. [pm] and [nd].
	// These values are read periodically.
	// Values are normally huge, e.g. pos=18000000000 [nd].
	//
	{attribute 'OPC.UA.DA' := '0'}
	devStatus:			T_SA_DEV_STATUS; 

END_STRUCT
END_TYPE

// ---- GVLs/GVL_Cryo_Temperatures.TcGVL
{attribute 'qualified_only'}
VAR_GLOBAL
	
// Temperature Sensors
	{attribute 'OPC.UA.DA' := '1'}
	Temp_1 : REAL;
	
	{attribute 'OPC.UA.DA' := '1'}
	Temp_2 : REAL;

	{attribute 'OPC.UA.DA' := '1'}
	Temp_3 : REAL;

	{attribute 'OPC.UA.DA' := '1'}
	Temp_4 : REAL;	
	
// Heater 

	{attribute 'OPC.UA.DA' := '1'}
	CryoHeater_1 : UINT;
	
	{attribute 'OPC.UA.DA' := '1'}
	CryoHeater_2 : UINT;
	
	{attribute 'OPC.UA.DA' := '1'}
	CryoHeater_3 : UINT;
END_VAR

// ---- GVLs/GVL_DL_Scanning_Homming.TcGVL
{attribute 'qualified_only'}
VAR_GLOBAL
	{attribute 'OPC.UA.DA':='1'}
	bHomming :BOOL;
	
	{attribute 'OPC.UA.DA':='1'}
	sHommingStatus :STRING;
	
	{attribute 'OPC.UA.DA':='1'}
	bTrigCameraImages :BOOL;
END_VAR

// ---- POUs/CameraTrig.TcPOU
PROGRAM CameraTrig
VAR
bCameraIN_1 AT %I* : BOOL;

bCameraIN_2 AT %I* : BOOL;

bCameraOUT_1 AT %Q* : BOOL;

bCameraOUT_2 AT %Q* : BOOL;

{attribute 'OPC.UA.DA':='1'}
b_Camera_in_1 :BOOL;
{attribute 'OPC.UA.DA':='1'}
b_Camera_in_2 :BOOL;
{attribute 'OPC.UA.DA':='1'}
b_Camera_out_1 :BOOL;
{attribute 'OPC.UA.DA':='1'}
b_Camera_out_2 :BOOL;
END_VAR

b_Camera_in_1 :=   bCameraIN_1; 

b_Camera_in_2 :=   bCameraIN_2; 

 bCameraOUT_1 :=  b_Camera_out_1;

 bCameraOUT_2 :=  b_Camera_out_2;

END_PROGRAM

// ---- POUs/MAIN.TcPOU
PROGRAM MAIN
VAR



// DL Servo
	
{attribute 'OPC.UA.DA':='1'}

DL_Servo_1: FB_MOTOR;

// DL Newport stepper
	
{attribute 'OPC.UA.DA':='1'}
DL_2: FB_MOTOR;

// Camera triggers

//bCameraIN_1 AT %I* : BOOL;

//bCameraIN_2 AT %I* : BOOL;

//bCameraOUT_1 AT %Q* : BOOL;

//bCameraOUT_2 AT %Q* : BOOL;

//{attribute 'OPC.UA.DA':='1'}
//b_Camera_in_1 :BOOL;
//{attribute 'OPC.UA.DA':='1'}
//b_Camera_in_2 :BOOL;
//{attribute 'OPC.UA.DA':='1'}
//b_Camera_out_1 :BOOL;
//{attribute 'OPC.UA.DA':='1'}
//b_Camera_out_2 :BOOL;

{attribute 'OPC.UA.DA':='1'}
fbCryoState : FB_Cryostat_State;

// Homming
iLocalCOntrolStatus : INT;


//Fring Scanning

// Time Stamp
fbGetSystemTime  : GETSYSTEMTIME;
fileTime         : T_FILETIME;
{attribute 'OPC.UA.DA':='1'}
sTime            : STRING;

// NPT PTP

time_info:	FB_TIME;

///

// Filter Wheel

FILTER_WHEEL	:	FB_SCIFY_FILTER_WHEEL_FW102C;

// Accelerometer

in_nVib_X AT %I* :DINT;	
in_nVib_Y AT %I* :DINT;
in_nVib_Z AT %I* :DINT;

{attribute 'OPC.UA.DA':='1'}
nVib_X:	DINT;
{attribute 'OPC.UA.DA':='1'}
nVib_Y:	DINT;
{attribute 'OPC.UA.DA':='1'}
nVib_Z:	DINT;

////
//Shutters
//////
{attribute 'OPC.UA.DA':='1'}
shutter_1:		FB_SHUTTER;


/// Tip-tilt motors
{attribute 'OPC.UA.DA':='1'}
tiptilt_1: FB_MOTOR;




END_VAR


fbCryoState();

DL_Servo_1(sName:='DL_Servo_1', nNOVRAM_DevId:=5, nNOVRAM_Offset:= 1000);

DL_2(sName:='DL_2_Newport', nNOVRAM_DevId:=5, nNOVRAM_Offset:= 2000);

//bCameraOUT_1 := GVL_DL_Scanning_Homming.bTrigCameraImages;


// Time Stamps

fbGetSystemTime(timeLoDW=>fileTime.dwLowDateTime, timeHiDW=>fileTime.dwHighDateTime );
sTime := SYSTEMTIME_TO_STRING( FILETIME_TO_SYSTEMTIME( fileTime ) );

time_info();

// Filter Wheel

FILTER_WHEEL(in_bSimulation:= FALSE, in_sName:= 'FILTER_WHEEL', in_nPeriod:= 1200);

// Vibration from Accelero sensor

nVib_X := in_nVib_X;
nVib_Y := in_nVib_Y;
nVib_Z := in_nVib_Z;

////  Shutters

shutter_1(
	in_sName:= 'Shutter_1', 
	in_bActiveLowClosed:= , 
	in_bActiveLowFault:= , 
	in_bActiveLowOpen:= TRUE, 
	in_bActiveLowSwitch:= , 
	in_bIgnoreClosed:= , 
	in_bIgnoreFault:= , 
	in_bIgnoreOpen:= , 
	in_bInitialState:= , 
	in_nTimeout:= , 
	in_bLogExtTime:= , 
	in_bLog:= );
	
/// Tip-tilt motors

tiptilt_1(sName:='Tip-Tilt_1', nNOVRAM_DevId:=5, nNOVRAM_Offset:= 4000);


//b_Camera_in_1 :=   bCameraIN_1; 

//b_Camera_in_2 :=   bCameraIN_2; 

//b_Camera_out_1 :=  bCameraOUT_1;

//b_Camera_out_2 :=  bCameraOUT_2;

END_PROGRAM

// ---- POUs/FB_Cryostat_State.TcPOU
FUNCTION_BLOCK FB_Cryostat_State
VAR_INPUT
END_VAR
VAR_OUTPUT
END_VAR
VAR
	nCryotemp_1 AT %I* : INT;
	nCryotemp_2 AT %I* : INT;
	nCryotemp_3 AT %I* : INT;
	nCryotemp_4 AT %I* : INT;
	
	nCryoHeater_1 AT %Q* : UINT;
	nCryoHeater_2 AT %Q* : UINT;
	nCryoHeater_3 AT %Q* : UINT;
END_VAR

GVL_Cryo_Temperatures.Temp_1 := nCryotemp_1 /10;

GVL_Cryo_Temperatures.Temp_2 := nCryotemp_2 /10;

GVL_Cryo_Temperatures.Temp_3 := nCryotemp_3 /10;

GVL_Cryo_Temperatures.Temp_4 := nCryotemp_4 /10;

nCryoHeater_1 := GVL_Cryo_Temperatures.CryoHeater_1;
nCryoHeater_1 := GVL_Cryo_Temperatures.CryoHeater_2;
nCryoHeater_1 := GVL_Cryo_Temperatures.CryoHeater_3;

END_FUNCTION_BLOCK

// ---- POUs/FILTER_WHEEL/FB_SCIFY_FILTER_WHEEL_FW102C.TcPOU
FUNCTION_BLOCK FB_SCIFY_FILTER_WHEEL_FW102C EXTENDS FB_RS_BASE
VAR_INPUT
	{attribute 'OPC.UA.DA' := '0'}
	in_nPeriod:	DINT := 10000;	// Interval for periodic reading [ms], default 10000 ms = 10 sec 
END_VAR
VAR_OUTPUT
END_VAR
VAR CONSTANT
	{attribute 'OPC.UA.DA' := '0'}
	//sCmdSuffix:		STRING(16) := '$0D$0A'; // CR LF
	sCmdSuffix:		STRING(16) := '$0D';		// CR
	{attribute 'OPC.UA.DA' := '0'}
	sReplySuffix:	STRING(16) := '$3E';		// >
END_VAR
VAR
	{attribute 'OPC.UA.DA' := '1'}
	cfg:		T_SCIFY_FILTER_WHEEL_CFG;		//  Config parameters
	{attribute 'OPC.UA.DA' := '1'}
	ctrl:		T_JANSSEN_CTRL;					//  Control parameters
	{attribute 'OPC.UA.DA' := '1'}
	{attribute 'OPC.UA.DA.Access' := '1'}
	info:		T_JANSSEN_INFO; 				//  Info parameters - ReadOnly
	{attribute 'OPC.UA.DA' := '1'}
	{attribute 'OPC.UA.DA.Access' := '1'}
	stat:		T_SCIFY_FILTER_WHEEL_STAT;					//  Status parameters - ReadOnly
	{attribute 'OPC.UA.DA' := '1'}
	ch_ctrl:	T_JANSSEN_CH_CTRL;				//  Channel control

	{attribute 'OPC.UA.DA' := '0'}
	comm:		FB_RS_COMM_NO_SIM;					// Instance of generic comm object. OPC UA Disabled!!!
	
	//{attribute 'OPC.UA.DA' := '0'}
	//comm:		FB_RS_COMM_LAKESHORE;	// Instance of Lakeshore customized comm 
	
	(* Pointers *)
	{attribute 'OPC.UA.DA' := '0'}
	ptrCommCfg:		POINTER TO T_RS_COMM_CFG 	:= ADR(comm.cfg);	(* Pointer to comm.cfg instance *)
	{attribute 'OPC.UA.DA' := '0'}
	ptrCommCtrl:	POINTER TO T_RS_COMM_CTRL 	:= ADR(comm.ctrl);	(* Pointer to comm.ctrl instance *)
	{attribute 'OPC.UA.DA' := '0'}
	ptrCommStat:	POINTER TO T_RS_COMM_STAT 	:= ADR(comm.stat);	(* Pointer to comm.stat instance *)
	{attribute 'OPC.UA.DA' := '0'}
	ptrInitCmds:	POINTER TO ARRAY [1..4] OF T_JANSSEN_COMMAND;		(* Pointer to INIT commands *)
	{attribute 'OPC.UA.DA' := '0'}
	ptrReadCmds:	POINTER TO ARRAY [1..4] OF T_JANSSEN_COMMAND;		(* Pointer to READ commands *)


	(* Timers *)
	{attribute 'OPC.UA.DA' := '0'}
	fbTimer:			TON; (* General Timeout *)
	
	(* Misc internal vars *)
	{attribute 'OPC.UA.DA' := '0'}
	cmdCounter:			INT := 1;

END_VAR

// Set references
cfgRef	REF=cfg;
ctrlRef	REF=ctrl;
statRef	REF=stat;


(* Execute comm instance *)
comm(in_sCmdSuffix:=sCmdSuffix, in_sReplySuffix:=sReplySuffix, in_nTimeout:=3000);



// Execute the base class object FB_RS_BASE
SUPER^();

METHOD ActivityInitializing
VAR_INPUT
	bExecute:	BOOL;
END_VAR
VAR_INST
	{attribute 'OPC.UA.DA' := '0'}
    nMethodState:	INT := 0;	// State Machine current state
END_VAR

// SmarACT
SetAction('ActivityInitializing');


IF NOT bExecute THEN
	nMethodState	:= 0;	// Reset the state machine
	cmdCounter		:= -1;	// First init command. CASE 15: will increment it to 0
	//cmdCounter		:= 1;	
	RETURN;
END_IF

// Handle State Machine
CASE nMethodState OF
	0:	// Initialize COMM port
		(* Reset the port *)
		ptrCommCtrl^.nCommand	:= E_RS_COMM_CMD.INIT;
		ptrCommCtrl^.bExecute	:= TRUE;

		(* Start the timer by going false/true *)
		fbTimer (IN := FALSE); (* Reset timer *)
		fbTimer (IN := TRUE, PT := T#5S); (* 5 sec timeout for reply *)

		nMethodState 	:= 15;	// On next cycle wait until the comm port is reset, i.e. idle
		
	15:	// Wait IDLE
		fbTimer (IN := TRUE);
		IF M_GetCommStatus() = E_RS_COMM_STATUS.IDLE  AND M_GetCommInitialised() THEN
			// Communication is IDLE 
			fbTimer (IN := FALSE);	// disable timer 
			stat.sReply		:= ptrCommStat^.sReply;	// Save the reply

			// Extract values from the reply to a stat variable.
			IF ptrCommCtrl^.bHasReply	THEN
				// Index is not important for INIT commands because they don't
				// refer to MODule or CHANnel.
				// We put zero for the input parameter.
				M_ReadReply();	// Index is not important for INIT commands.
			END_IF

			cmdCounter		:= cmdCounter + 1;	// Increment init command index
			fbTimer (IN := FALSE);	// disable timer 
			fbTimer (IN := TRUE, PT := cfg.tDelay_Init); // Wait INIT delay
			bCommProblem	:= FALSE;
			nMethodState 	:= 18;	// Execute next device INIT command
		ELSIF M_GetCommStatus() = E_RS_COMM_STATUS.ERROR  AND fbTimer.ET > T#4900MS THEN
			fbTimer (IN := FALSE);
			SetStatus(E_LAKESHORE_ERROR.COMM, 'ERROR: Communication error');	
			bCommProblem	:= TRUE;
			nEvent := E_SM_EVENT.ERRINIT;
			RETURN;
		ELSIF fbTimer.Q THEN
			// Timer expired after 5 sec. This is an error.
			fbTimer (IN := FALSE);
			SetStatus(E_LAKESHORE_ERROR.TIMEOUT, 'ERROR: Communication timeout');	
			bCommProblem	:= TRUE;
			nEvent := E_SM_EVENT.ERRINIT;
			RETURN;
		END_IF

	
	
	18:	// Wait INIT Delay
		fbTimer (IN := TRUE);
		IF fbTimer.Q THEN
			// Timer expired after 5 sec. This is an error.
			fbTimer (IN := FALSE);
			nMethodState 	:= 20;	// Execute next device INIT command
			RETURN;
		END_IF

	
	
	20:	// INIT DEV
		IF cfg.cmdList_Init[cmdCounter].cmd = '' THEN
			// Device INIT is done. Go to IDLE 
			stat.bInitialised 	:= TRUE;
			cmdCounter			:= 1;
			SetStatus(E_SM_ERROR.OK, 'IDLE');
			nEvent 		:= E_SM_EVENT.INITDONE;
			RETURN;
		END_IF
		
		(* Send INIT command with index cmdCounter *)
		ptrCommCtrl^.nCommand		:= E_RS_COMM_CMD.SEND;
		ptrCommCtrl^.sCmd			:= cfg.cmdList_Init[cmdCounter].cmd;
		ptrCommCtrl^.nNumReplies	:= cfg.cmdList_Init[cmdCounter].nReplies;
		ptrCommCtrl^.bHasReply		:= cfg.cmdList_Init[cmdCounter].nReplies > 0;
		ptrCommCtrl^.bExecute		:= TRUE;
	
		(* Start the timer by going false/true *)
		fbTimer (IN := FALSE); (* Reset timer *)
		fbTimer (IN := TRUE, PT := T#5S); (* 5 sec timeout for reply *)

		// On next cycle wait until the comm port is idle
		nMethodState 	:= 15;	// On next cycle wait until the comm port is idle
	
END_CASE

(*
// Lakeshore
SetAction('ActivityInitializing');


IF NOT bExecute THEN
	nMethodState	:= 0;	// Reset the state machine
	cmdCounter		:= 1;	// Init will start from the first init command
	RETURN;
END_IF

// Handle State Machine
CASE nMethodState OF
	0:	// Set communication parameters and Model configuration

		(* Set comm suffixes for commands and replies *)
		ptrCommCfg^.sCmdSuffix		:= sCmdSuffix;
		ptrCommCfg^.sReplySuffix	:= sReplySuffix;

		// Set monitoring period (input parameter)
		cfg.tDelay_Periodic	:= DINT_TO_TIME(in_nPeriod);
		// Auto monitor, i.e. monitor in Standby_Ready as well
		cfg.bAutoMonitor	:= TRUE; 
		//cfg.bAutoMonitor	:= FALSE;

		(* Set pointer to INIT and READ commands *)
		ptrInitCmds := ADR(cfg.cmdList_Init);
		//ptrReadCmds := ADR(cfg.cmdList_Read);
		ptrReadCmds := ADR(cfg.cmdList_Mon);
		(* Set initial state and status *)
		stat.bInitialised	:= FALSE;
		stat.sReply			:= '';
		stat.sDeviceID		:= '';

		SetStatus(E_SM_ERROR.OK, 'BUSY');

		nMethodState := 10;				// Go to next state, i.e. INIT_COMM

	10:	// Initialize COMM port
		(* Reset the serial port *)
		ptrCommCtrl^.nCommand	:= E_RS_COMM_CMD.INIT;
		ptrCommCtrl^.bExecute	:= TRUE;

		// Init dev will start from the first init command.
		// We set counter to 0. It will be incremented in Wait IDLE.
		cmdCounter	:= 0;

		(* Start the timer by going false/true *)
		fbTimer (IN := FALSE); (* Reset timer *)
		fbTimer (IN := TRUE, PT := T#5S); (* 5 sec timeout for reply *)

		nMethodState 	:= 15;	// On next cycle wait until the comm port is reset, i.e. idle
		
	15:	// Wait IDLE
		fbTimer (IN := TRUE);
		IF comm.stat.nStatus = E_RS_COMM_STATUS.IDLE THEN
			// Communication is IDLE 
			fbTimer (IN := FALSE);	// disable timer 
			 stat.sReply		:= ptrCommStat^.sReply;	// Save the reply
			(*
			IF cmdCounter >= 1 THEN
				// We are IDLE after an INIT command, i.e. CCC_CMD_RESET or CCC_CMD_GET_VERS
				IF ptrInitCmds^ [cmdCounter].cmd = cfg.CCC_CMD_RESET  THEN
					(* No action. Just check proper reply. *)
					IF FIND (stat.sReply, 'N')= 1 THEN
						SetStatus(E_CCC_ERROR.COMM, 'ERROR: Failed to RESET device');
						bCommProblem	:= TRUE;
						nEvent := E_SM_EVENT.ERRINIT;
						RETURN;
					END_IF
				ELSIF ptrInitCmds^ [cmdCounter].cmd = cfg.CCC_CMD_GET_VERS  THEN
					(* Save the reply into stat.sDeviceID. *)
					IF FIND (stat.sReply, 'N')= 1 THEN
						SetStatus(E_CCC_ERROR.COMM, 'ERROR: Command GET_VERS failed');
						bCommProblem	:= TRUE;
						nEvent := E_SM_EVENT.ERRINIT;
						RETURN;
					ELSIF FIND (stat.sReply, 'ESO')<> 2 THEN
						SetStatus(E_CCC_ERROR.COMM, 'ERROR: Failed to get device ID');
						bCommProblem	:= TRUE;
						nEvent := E_SM_EVENT.ERRINIT;
						RETURN;
					ELSE
						stat.sDeviceID	:= MID (stat.sReply, LEN(stat.sReply)-5, 2);
					END_IF
				END_IF
			END_IF
			*)
			// Restart the timer for delay between INIT commands
			fbTimer (IN := FALSE);	// disable timer 
			
			fbTimer (IN := TRUE, PT := cfg.tDelay_Init); // Wait INIT delay
			
			cmdCounter		:= cmdCounter + 1;	// Increment init command index
			bCommProblem	:= FALSE;
			nMethodState 	:= 18;	// Execute next device INIT command
		ELSIF comm.stat.nStatus = E_RS_COMM_STATUS.ERROR THEN
			fbTimer (IN := FALSE);
			SetStatus(E_CCC_ERROR.COMM, 'ERROR: Communication error');	
			bCommProblem	:= TRUE;
			nEvent := E_SM_EVENT.ERRINIT;
			RETURN;
		ELSIF fbTimer.Q THEN
			// Timer expired after 5 sec. This is an error.
			fbTimer (IN := FALSE);
			SetStatus(E_JANSSEN_ERROR.TIMEOUT, 'ERROR: Communication timeout');	
			bCommProblem	:= TRUE;
			nEvent := E_SM_EVENT.ERRINIT;
			RETURN;
		END_IF 

	
	
	18:	// Wait INIT Delay
		fbTimer (IN := TRUE);
		IF fbTimer.Q THEN
			// Timer expired after 5 sec. This is an error.
			fbTimer (IN := FALSE);
			nMethodState 	:= 20;	// Execute next device INIT command
			RETURN;
		END_IF

	
	
	20:	// INIT DEV
		IF ptrInitCmds^ [cmdCounter].cmd = '' THEN
			// Device INIT is done. Go to IDLE 
			stat.bInitialised 	:= TRUE;
			cmdCounter			:= 1;
			SetStatus(E_JANSSEN_STATUS.IDLE, 'IDLE');
			nEvent 		:= E_SM_EVENT.INITDONE;
			RETURN;
		END_IF
		
		
		
		(* Send INIT command with index cmdCounter *)
		ptrCommCtrl^.nCommand		:= E_RS_COMM_CMD.SEND;
		ptrCommCtrl^.sCmd			:= ptrInitCmds^ [cmdCounter].cmd;
		ptrCommCtrl^.nNumReplies	:= 1;
		ptrCommCtrl^.bHasReply		:= TRUE;
		ptrCommCtrl^.bExecute		:= TRUE;
	
		(* Start the timer by going false/true *)
		fbTimer (IN := FALSE); (* Reset timer *)
		fbTimer (IN := TRUE, PT := T#5S); (* 5 sec timeout for reply *)
		
		// On next cycle wait until the comm port is idle
		nMethodState 	:= 15;	// On next cycle wait until the comm port is idle
	
END_CASE
*)
END_METHOD

METHOD ActivityMonitoring
VAR_INPUT
	bExecute:	BOOL;
END_VAR
VAR_INST
	{attribute 'OPC.UA.DA' := '0'}
    nMethodState:	INT := 0;	// State Machine current state
	{attribute 'OPC.UA.DA' := '0'}
	nRetries:		INT := 0;	// Number of retries in case of communication problems
	
	{attribute 'OPC.UA.DA' := '0'}
	nCmdType:		E_JANSSEN_CMD_TYPE := E_JANSSEN_CMD_TYPE.READ;
	{attribute 'OPC.UA.DA' := '0'}
	devCmd:			T_JANSSEN_COMMAND;	// Device command to be sent
	
	{attribute 'OPC.UA.DA' := '0'}
	nCmdIdx:		UINT := 0;	// Command index in specific command list. [0..15]

END_VAR
VAR
	bError:			BOOL;
	
END_VAR

//SmarACT
//
// At least one module must be used.
// If not, don't do anything.
//
(*
IF stat.nNumMod = 0	THEN
	SetAction('ERROR: No Module Used !!!'); 
	SetStatus(E_SM_ERROR.INIT_FAILURE, 'ERROR: No Module Used !!!');
	RETURN;
END_IF
*)
IF NOT cfg.bAutoMonitor AND stat.nSubstate = E_RS_BASE_SUBSTATE.NOTOP_READY THEN
	SetAction('No Monitoring'); 
	SetStatus(E_SM_ERROR.OK, 'IDLE');
	nMethodState	:= 0;	// Reset the state machine
	RETURN;
END_IF

IF NOT bExecute THEN
	SetAction('ActivityMonitoring'); 
	SetStatus(E_SM_ERROR.OK, 'BUSY');
	nMethodState	:= 0;	// Reset the state machine
	nCmdType		:= E_JANSSEN_CMD_TYPE.READ;	// We start with READ commands.
	RETURN;
END_IF

// Handle State Machine
CASE nMethodState OF
	0:	// Get valid channel.
		// This call will check if the current channel is used.
		// If not, it will take next available channel.
		
		//nChIdx	:= M_GetValidChannel(nChIdx);
		
		
		
		// If this is the very first command for the channel,
		// Set commands.
		IF nCmdIdx = 0	THEN
			M_SetCmdList();
		END_IF
		
		
		// Get next command to execute.
		// The command depends on the state of the positioner and 
		// the current index (nCmdIdx) of the command in the list.
		//
		//devCmd	:= M_GetCommand(nCmdIdx);
		devCmd	:= M_GetCommand(nCmdIdx);
			
		// Check if we have arrived at the end of the command list.
		// In this case, go to the next channel.
		IF devCmd.cmd = '' THEN
			// We have executed all commands.
			// Check if we have to exit Monitoring
			IF nNextState <> E_RS_BASE_STATE.NONE	THEN
				SetStatus(E_SM_ERROR.OK, nNextDescription);
				SetState(nNextState, nNextSubstate);
				nNextState		:= E_RS_BASE_STATE.NONE;
				nNextSubstate	:= E_RS_BASE_SUBSTATE.NONE;
				nNextDescription:= '';
				RETURN;
			END_IF
			
			//
			// Update Positioner status
			//
			//ptrCH[nChIdx]^.M_UpdateStatus();
			
			//M_UpdateStatus();
			
			// Check if the State Machine State should be changed.
			// If yes, M_SetNextPosState() will set new state and return TRUE.
			// This can happen due to any Positioner control command (CAL, REF, RESET, ENABLE, DISABLE, MOVE or STOP)
			//IF ptrCH[nChIdx]^.M_SetNextPosState()	THEN
			
			IF M_SetNextPosState()	THEN
				// The State has changed.
				// Reset command index to 0, i.e. start from the first command.
				nCmdIdx	:= 0;
			//ELSE
				// Get NEXT valid channel
				//nChIdx	:= M_GetValidChannel(nChIdx + 1);
				
				// Reset command index to 0
				//nCmdIdx	:= 0;
			END_IF
					
				
			// Wait tDelay_Periodic before re-starting the READ.
			SetStatus(E_SM_ERROR.OK, 'IDLE');
			
			(* Start the timer by going false/true *)
			fbTimer (IN := FALSE); (* Reset timer *)
			fbTimer (IN := TRUE, PT := cfg.tDelay_Periodic);
			nMethodState 	:= 10;	// Goto Wait for tDelay_Periodic
			RETURN;
		END_IF
		
		// Send command
		ptrCommCtrl^.nCommand		:= E_RS_COMM_CMD.SEND;
		ptrCommCtrl^.sCmd			:= devCmd.cmd;
		ptrCommCtrl^.nNumReplies	:= devCmd.nReplies;
		ptrCommCtrl^.bHasReply		:= devCmd.nReplies > 0;
		ptrCommCtrl^.bExecute		:= TRUE;
		
		
		
		statRef.sErrorText	:= 'BUSY';

		// In case we are executing a CTRL command with no replies,
		// we apply a long timeout.
		// However, when the comm port becomes IDLE and after at 
		// least 200ms, we go to the next command. (see nMethodState 12:)
		IF NOT ptrCommCtrl^.bHasReply THEN
			fbTimer (IN := FALSE); // Reset timer
			fbTimer (IN := TRUE, PT := T#10S); 
			nCmdIdx			:= nCmdIdx + 1;	// Go to next command.
			nMethodState	:= 12;				// Goto WAIT for delay
			RETURN;
		ELSE			
			// There is a reply, i.e. this is a 'READ' command.
			// For regular READ commands, apply short delay of 10ms before 
			// checking the status of comm port. 
			// Start the timer by going false/true
			fbTimer (IN := FALSE); // Reset timer
			fbTimer (IN := TRUE, PT := T#10MS);	

			statRef.sErrorText	:= 'BUSY';
			nMethodState := 15;	// Goto short delay
			RETURN;
		END_IF
		
		
		
	10:	// Wait until the delay timeout expires
		fbTimer (IN := TRUE);

		(* If Timer has expired, go to the next state. *)
		IF fbTimer.Q THEN
			fbTimer (IN := FALSE);
			nMethodState 	:= 0;				// Goto handling of next command
			RETURN;
		END_IF
	
	12:	// Wait until the comm port is idle and at least 200ms have expired.
		// Otherwise, wait the PT period.
		fbTimer (IN := TRUE);

		IF (M_GetCommStatus() = E_RS_COMM_STATUS.IDLE  AND  fbTimer.ET > T#200MS)	OR
			fbTimer.Q	THEN
			fbTimer (IN := FALSE);
			nMethodState 	:= 0;				// Goto handling of next command
			RETURN;
		END_IF

	
	15:	// Wait until the delay timeout expires
		fbTimer (IN := TRUE);

		(* If Timer has expired, go to the next state. *)
		IF fbTimer.Q THEN
			fbTimer (IN := FALSE);
			fbTimer (IN := TRUE, PT := T#3S);	// 3 sec timeout for reply
			statRef.sErrorText	:= 'BUSY';
			nMethodState 	:= 20;	// Goto Wait for IDLE/Reply
			RETURN;
		END_IF
	



	20:	// Wait for the reading to complete, i.e. IDLE
		fbTimer (IN := TRUE);
		IF M_GetCommStatus() = E_RS_COMM_STATUS.IDLE THEN
			// Communication is IDLE 
			fbTimer (IN := FALSE);	// disable timer 
			stat.sReply		:= ptrCommStat^.sReply;	// Save the reply
			
			// Extract values from the reply to a stat variable.
			M_ReadReply();

			bCommProblem	:= FALSE;
			nRetries		:= 0;	// Reset number of retries

			nCmdIdx			:= nCmdIdx + 1;	// Go to next command.
			
			nMethodState 	:= 0;				// Goto Send command
			nEvent := E_SM_EVENT.COMMOK;
			RETURN;
		ELSIF M_GetCommStatus() = E_RS_COMM_STATUS.ERROR OR fbTimer.Q THEN
			fbTimer (IN := FALSE);
			SetStatus(E_LAKESHORE_ERROR.COMM, 'ERROR: Communication error');	
			bCommProblem	:= TRUE;
			// Retry up to 2 times
			nRetries		:= nRetries + 1;		// Increment number of retries
			stat.nRetries	:= stat.nRetries + 1;	// Increment total number of retries
			IF nRetries > 1 THEN
				nEvent := E_SM_EVENT.ERRCOMM;
				RETURN;
			END_IF
			// Apply a short delay of 1 sec and retry
			fbTimer (IN := FALSE); (* Reset timer *)
			fbTimer (IN := TRUE, PT := T#1000MS);
			nMethodState := 10;				// Goto Wait 
			RETURN;
		END_IF

	
END_CASE

(*

// Lakeshore
IF NOT bExecute THEN
	SetAction('ActivityMonitoring'); 
	SetStatus(E_SM_ERROR.OK, 'BUSY');
	nMethodState	:= 0;	// Reset the state machine
	cmdCounter		:= 1;	// Reading will start from the first command in the array
	nCmdType		:= E_JANSSEN_CMD_TYPE.READ;	// We start with READ commands.
	nRetries		:= 0;					
	RETURN;
END_IF

// Handle State Machine
CASE nMethodState OF
	0:	// Execute a command from the command array
		IF ptrReadCmds^ [cmdCounter].cmd = '' OR cmdCounter > 4 THEN
			// We arrived to the end of the array of pre-defined commands
			// Check if we have to exit Monitoring
			IF nNextState <> E_RS_BASE_STATE.NONE	THEN
				SetStatus(E_SM_ERROR.OK, nNextDescription);
				SetState(nNextState, nNextSubstate);
				nNextState		:= E_RS_BASE_STATE.NONE;
				nNextSubstate	:= E_RS_BASE_SUBSTATE.NONE;
				nNextDescription:= 'IDLE';
				RETURN;
			END_IF

			// Periodic READ is done. Wait tDelay_Periodic before re-starting the READ.
			cmdCounter	:= 1;
			SetStatus(E_SM_ERROR.OK, 'IDLE');
			
			(* Start the timer by going false/true *)
			fbTimer (IN := FALSE); (* Reset timer *)
			fbTimer (IN := TRUE, PT := cfg.tDelay_Periodic);
			nMethodState := 10;				// Goto Wait for tDelay_Periodic
			RETURN;
		END_IF
		
		(* Send command with index cmdCounter *)
		ptrCommCtrl^.nCommand		:= E_RS_COMM_CMD.SEND;
		ptrCommCtrl^.sCmd			:= ptrReadCmds^ [cmdCounter].cmd;
		ptrCommCtrl^.nNumReplies	:= 1;
		ptrCommCtrl^.bHasReply		:= TRUE;
		ptrCommCtrl^.bExecute		:= TRUE;
		
		stat.sErrorText := 'BUSY';
		(* Start the timer by going false/true *)
		fbTimer (IN := FALSE); (* Reset timer *)
		fbTimer (IN := TRUE, PT := T#5S); (* 5 sec timeout for reply *)

		nMethodState := 20;				// Goto WAIT for Reading to complete,

	10:	// Wait until the delay timeout expires
		fbTimer (IN := TRUE);

		// Check if we have to exit Monitoring
		IF nNextState <> E_RS_BASE_STATE.NONE THEN
			fbTimer (IN := FALSE); (* Stop the timer *)
			SetStatus(E_SM_ERROR.OK, nNextDescription);
			SetState(nNextState, nNextSubstate);
			nNextState		:= E_RS_BASE_STATE.NONE;
			nNextSubstate	:= E_RS_BASE_SUBSTATE.NONE;
			nNextDescription:= 'IDLE';
			RETURN;
		END_IF
	
		(* If Timer has expired, go to the next state. *)
		IF fbTimer.Q THEN
			fbTimer (IN := FALSE);
			cmdCounter		:= 1;	// Reading will start from the first command in the array
			nMethodState 	:= 0;	// Goto Wait for tDelay_Periodic
			RETURN;
		END_IF
	


	20:	// Wait for the reading to complete, i.e. IDLE
		fbTimer (IN := TRUE);
		IF comm.stat.nStatus = E_RS_COMM_STATUS.IDLE THEN
			bError	:= FALSE;
			// Communication is IDLE 
			fbTimer (IN := FALSE);	// disable timer 
			stat.sReply		:= ptrCommStat^.sReply;	// Save the reply
			 
			M_ReadReply();
		//IF ptrCommCtrl^.sCmd = '/GBR RS422' THEN
			// Get the DEVice ID
			//stat.sBaud_rate_RS422	:= LEFT(stat.sReply, LEN(stat.sReply) - LEN(sReplySuffix));
		//END_IF
			(*
			(* Extract the readins from the reply. *)
			IF ptrReadCmds^ [cmdCounter].cmd = cfg.CCC_CMD_GET_STAT  THEN
				IF NOT M_UpdateDevStatus() THEN
					SetStatus(E_CCC_ERROR.COMM, 'ERROR: GET_STAT reply format not correct');
					bError	:= TRUE;
				END_IF
			ELSIF ptrReadCmds^ [cmdCounter].cmd = cfg.CCC_CMD_GET_TEMP  THEN
				IF NOT M_UpdateDevTemps() THEN
					SetStatus(E_CCC_ERROR.COMM, 'ERROR: GET_TEMP reply format not correct');
					bError	:= TRUE;
				END_IF
			ELSIF ptrReadCmds^ [cmdCounter].cmd = cfg.CCC_CMD_GET_FLOW  THEN
				IF NOT M_UpdateDevFlows() THEN
					SetStatus(E_CCC_ERROR.COMM, 'ERROR: GET_FLOW reply format not correct');
					bError	:= TRUE;
				END_IF
			END_IF
			*)
			bCommProblem	:= FALSE;
			nRetries		:= 0;	// Reset number of retries
			
			// Check if we have to exit Monitoring
			IF nNextState <> E_RS_BASE_STATE.NONE THEN
				fbTimer (IN := FALSE); (* Stop the timer *)
				SetStatus(E_SM_ERROR.OK, nNextDescription);
				SetState(nNextState, nNextSubstate);
				nNextState		:= E_RS_BASE_STATE.NONE;
				nNextSubstate	:= E_RS_BASE_SUBSTATE.NONE;
				nNextDescription:= 'IDLE';
				RETURN;
			END_IF
	
			cmdCounter		:= cmdCounter + 1;	// Reading will start from the first command in the array
			
			nMethodState 	:= 0;				// Goto Send command
			nEvent := E_SM_EVENT.COMMOK;
			RETURN;
		ELSIF comm.stat.nStatus = E_RS_COMM_STATUS.ERROR OR fbTimer.Q THEN
			fbTimer (IN := FALSE);
			SetStatus(E_JANSSEN_ERROR.COMM, 'ERROR: Communication error');	
			bCommProblem	:= TRUE;
			// Retry up to 2 times
			nRetries		:= nRetries + 1;		// Increment number of retries
			stat.nRetries	:= stat.nRetries + 1;	// Increment total number of retries
			IF nRetries > 1 THEN
				nEvent := E_SM_EVENT.ERRCOMM;
			END_IF
			// Apply a short delay of 1 sec and retry
			fbTimer (IN := FALSE); (* Reset timer *)
			fbTimer (IN := TRUE, PT := T#1000MS);
			nMethodState := 10;				// Goto Wait 
			RETURN;
		ELSIF bError THEN
			// Apply a short delay of 3 sec and retry
			fbTimer (IN := FALSE); (* Reset timer *)
			fbTimer (IN := TRUE, PT := T#3000MS);
			nMethodState := 10;				// Goto Wait 
			RETURN;
		END_IF

	
END_CASE
*)
END_METHOD

METHOD M_GetCalibrationValues : BOOL
(* FB to extract 'n' values from 'str' and copy them into stat.lrArrReadings starting from index 'idx'.*)

VAR_INPUT
	//idx:	INT;		(* arr [idx] will hold the first extracted value, arr [idx+1] the second one, etc. *)
	//n:		INT;		(* Number of values to extract from the string - command specific *)
	
	str:	STRING(255);		(* String returned in Lakeshore reply *)
	ch_idx:	INT;
END_VAR
VAR_OUTPUT
	ok:		BOOL;		(* TRUE if the reading was correct, i.e. 'n' values successfully extracted from 'str'.  *)
END_VAR

VAR
	idx:	INT := 1; // starting index
	n:		INT	:= 3; // Max values in Get calibration string
	i:		INT; 
	str_l:	STRING(255);
	pos:	INT;
	
	nCalibrationValues: ARRAY[1..3] OF DINT; 
END_VAR
i	:= 0;
str_l	:= str;
ok	:= TRUE; (* OK *)


WHILE i < n DO
	nCalibrationValues[idx + i]	:= STRING_TO_DINT(str_l); (* take the first number *)
	(* move to just after the comma *)
	IF i < (n-1) THEN
		pos := FIND (str_l, ','); (* find the comma *)
		IF pos = 0 THEN (* less than 'n' numbers present in the string *)
			ok	:= FALSE; (* ERROR *)
			i 	:= n;
		ELSE
			str_l := RIGHT (str_l, LEN(str_l) - pos);
			i	:= i + 1;
		END_IF
	ELSE
		i	:= i + 1;
	END_IF
END_WHILE

IF ch_idx = 1 THEN
	stat.nCalibrationValues_Cannel_1.nGainSetting:= nCalibrationValues[1];
	stat.nCalibrationValues_Cannel_1.nUpperThresholdValue:= nCalibrationValues[2];
	stat.nCalibrationValues_Cannel_1.nLowerThresholdValue:= nCalibrationValues[3];
ELSIF ch_idx = 2 THEN
	stat.nCalibrationValues_Cannel_2.nGainSetting:= nCalibrationValues[1];
	stat.nCalibrationValues_Cannel_2.nUpperThresholdValue:= nCalibrationValues[2];
	stat.nCalibrationValues_Cannel_2.nLowerThresholdValue:= nCalibrationValues[3];
ELSIF ch_idx = 3 THEN
	stat.nCalibrationValues_Cannel_3.nGainSetting:= nCalibrationValues[1];
	stat.nCalibrationValues_Cannel_3.nUpperThresholdValue:= nCalibrationValues[2];
	stat.nCalibrationValues_Cannel_3.nLowerThresholdValue:= nCalibrationValues[3];
END_IF
END_METHOD

//
// Get command with index 'index' from ctrl.cmdList[]
//
METHOD M_GetCommand : T_JANSSEN_COMMAND
VAR_INPUT
	index:		UINT;
END_VAR
VAR
	emptyCmd:	T_JANSSEN_COMMAND;
END_VAR
IF index < 0 OR index > 15	THEN
	// The index is not valid. Set empty command.
	M_GetCommand	:= emptyCmd;
ELSE
	M_GetCommand	:= ctrl.cmdList[index];
END_IF
END_METHOD

METHOD M_GetCommInitialised : BOOL
VAR_INPUT
END_VAR
// This is just a dummy method for BASE FB
M_GetCommInitialised	:= comm.M_GetInitialised();
END_METHOD

METHOD M_GetCommStatus : E_RS_COMM_STATUS
VAR_INPUT
END_VAR
M_GetCommStatus	:= comm.M_GetStatus();
END_METHOD

METHOD M_GetCounterValues : BOOL
(* FB to extract 'n' values from 'str' and copy them into stat.lrArrReadings starting from index 'idx'.*)

VAR_INPUT
	//idx:	INT;		(* arr [idx] will hold the first extracted value, arr [idx+1] the second one, etc. *)
	//n:		INT;		(* Number of values to extract from the string - command specific *)
	
	str:	STRING(255);		(* String returned in Lakeshore reply *)
	//ch_idx:	INT;
END_VAR
VAR_OUTPUT
	ok:		BOOL;		(* TRUE if the reading was correct, i.e. 'n' values successfully extracted from 'str'.  *)
END_VAR

VAR
	idx:	INT := 1; // starting index
	n:		INT	:= 4; // Max values in Get calibration string
	i:		INT; 
	str_l:	STRING(255);
	pos:	INT;
	
	nCounterValues: ARRAY[1..3] OF DINT; 
END_VAR
i	:= 0;
str_l	:= str;
ok	:= TRUE; (* OK *)


WHILE i < n DO
	nCounterValues[idx + i]	:= STRING_TO_DINT(str_l); (* take the first number *)
	(* move to just after the comma *)
	IF i < (n-1) THEN
		pos := FIND (str_l, ','); (* find the comma *)
		IF pos = 0 THEN (* less than 'n' numbers present in the string *)
			ok	:= FALSE; (* ERROR *)
			i 	:= n;
		ELSE
			str_l := RIGHT (str_l, LEN(str_l) - pos);
			i	:= i + 1;
		END_IF
	ELSE
		i	:= i + 1;
	END_IF
END_WHILE

stat.nCounterValue_Channel_1	:= nCounterValues[1];
stat.nCounterValue_Channel_2	:= nCounterValues[2];
stat.nCounterValue_Channel_3	:= nCounterValues[3];
END_METHOD

METHOD M_GetErrorString : STRING
VAR_INPUT
END_VAR
IF	stat.stState.bRANGE_LIMIT_REACHED		THEN
	M_GetErrorString	:= 'ERROR: Range limit reached';
ELSIF	stat.stState.bEND_STOP_REACHED	THEN
	M_GetErrorString	:= 'ERROR: End Stop reached';
ELSIF	stat.stState.bFOLLOWING_LIMIT_REACHED	THEN
	M_GetErrorString	:= 'ERROR: Following error';
ELSIF	stat.stState.bPOSITIONER_OVERLOAD		THEN
	M_GetErrorString	:= 'ERROR: Positioner overload';
ELSIF	stat.stState.bOVER_TEMPERATURE			THEN
	M_GetErrorString	:= 'ERROR: Overtemperature';
ELSIF	stat.stState.bPOSITIONER_FAULT			THEN
	M_GetErrorString	:= 'ERROR: Positioner fault';
ELSIF	stat.stState.bMOVEMENT_FAILED			THEN
	M_GetErrorString	:= 'ERROR: Movement failed';
ELSE
	M_GetErrorString	:= 'Positioner Error';
END_IF
END_METHOD

METHOD M_GetFailSafeState
VAR_INPUT
	sFailSafeState:		STRING;
END_VAR
 
IF FIND(sFailSafeState,'NO ERRORS PRESENT') > 0 THEN
	stat.stState.bControllerStateError := FALSE;
END_IF
END_METHOD

METHOD M_GetPositionControlStatus : BOOL
(* FB to extract 'n' values from 'str' and copy them into stat.lrArrReadings starting from index 'idx'.*)

VAR_INPUT
	//idx:	INT;		(* arr [idx] will hold the first extracted value, arr [idx+1] the second one, etc. *)
	//n:		INT;		(* Number of values to extract from the string - command specific *)
	str:	STRING(255);		(* String returned in Lakeshore reply *)
END_VAR
VAR_OUTPUT
	ok:		BOOL;		(* TRUE if the reading was correct, i.e. 'n' values successfully extracted from 'str'.  *)
END_VAR

VAR
	idx:	INT := 1; // starting index
	n:		INT	:= 8; // Max values in position control status string
	i:		INT; 
	str_l:	STRING(255);
	pos:	INT;
	
	nPositionContolStatusValues: ARRAY[1..8] OF DINT; 
END_VAR
i	:= 0;
str_l	:= str;
ok	:= TRUE; (* OK *)


WHILE i < n DO
	nPositionContolStatusValues[idx + i]	:= STRING_TO_DINT(str_l); (* take the first number *)
	(* move to just after the comma *)
	IF i < (n-1) THEN
		pos := FIND (str_l, ','); (* find the comma *)
		IF pos = 0 THEN (* less than 'n' numbers present in the string *)
			ok	:= FALSE; (* ERROR *)
			i 	:= n;
		ELSE
			str_l := RIGHT (str_l, LEN(str_l) - pos);
			i	:= i + 1;
		END_IF
	ELSE
		i	:= i + 1;
	END_IF
END_WHILE

stat.bPositionControl:= DINT_TO_BOOL(nPositionContolStatusValues[1]);
stat.bMovingToSetPoint:= DINT_TO_BOOL(nPositionContolStatusValues[2]);
stat.bInvalidSetPoint_1:= DINT_TO_BOOL(nPositionContolStatusValues[3]);
stat.bInvalidSetPoint_2:= DINT_TO_BOOL(nPositionContolStatusValues[4]);
stat.bInvalidSetPoint_3:= DINT_TO_BOOL(nPositionContolStatusValues[5]);

stat.nPositionError_1:= nPositionContolStatusValues[6];
stat.nPositionError_2:= nPositionContolStatusValues[7];
stat.nPositionError_3:= nPositionContolStatusValues[8];
END_METHOD

METHOD M_ReadReply : BOOL
VAR_INPUT
	//index:	UINT;	// Channel number!
END_VAR
VAR
	pos:			INT;	// Position of the terminator in the reply.
    parsed_reply: 	STRING;
	//refChStatus:	REFERENCE TO T_SA_CH_STATUS;
	length_reply: INT;
	length_suffix: INT;
	remaining_length: INT;
	
	////////////////////
	//Test String//////
	s_Test_String: STRING := '1,1,1,1,1,26,27,28';
	s_Test_Calibrstion_string: STRING := '74, 992, -56';
	//////////////////
END_VAR
//
// Reply should always end with in_sReplySuffix ('$R$N') character.
// Otherwise, it's an error.
// Only commands with the reply from which the value should be read are handled.
//

pos := FIND (stat.sReply, sReplySuffix);
length_suffix:= LEN(sReplySuffix);
length_reply:= LEN(stat.sReply);
remaining_length := length_reply - length_suffix;

IF pos > 0	THEN
	length_reply:= LEN(sReplySuffix);
	length_suffix:= LEN(stat.sReply);
	remaining_length := length_reply - length_suffix;
    parsed_reply := LEFT(stat.sReply, LEN(stat.sReply) - LEN(sReplySuffix));
	
	IF ptrCommCtrl^.sCmd = '*idn?' THEN
		// Get the DEVice ID
		stat.sDeviceID	:= parsed_reply;
	ELSIF ptrCommCtrl^.sCmd = 'pos?' THEN
		// Get the DEVice ID
		stat.nCurrentFilterPosition	:= parsed_reply;
	ELSIF ptrCommCtrl^.sCmd = 'speed?' THEN
		// Get the DEVice ID
		stat.bMoveSpeed	:= parsed_reply;
	ELSIF ptrCommCtrl^.sCmd = 'sensors?' THEN
		// Get the DEVice ID
		stat.bFilterSensors	:= parsed_reply;
	ELSIF ptrCommCtrl^.sCmd = 'baud?' THEN
		// Get the DEVice ID
		stat.sBaud_rate_RS232	:= parsed_reply;
	ELSIF ptrCommCtrl^.sCmd = 'STP 3' THEN
		// Get the DEVice ID
		stat.sChannel_3_Stop	:= parsed_reply;
	ELSIF ptrCommCtrl^.sCmd = 'GFS 1' THEN
		// Get the DEVice ID
		stat.sFailSafeState_1	:= parsed_reply;
		M_GetFailSafeState(parsed_reply);
	ELSIF ptrCommCtrl^.sCmd = 'GFS 2' THEN
		// Get the DEVice ID
		stat.sFailSafeState_2	:= parsed_reply;
	ELSIF ptrCommCtrl^.sCmd = 'GFS 3' THEN
		// Get the DEVice ID
		stat.sFailSafeState_3	:= parsed_reply;
	ELSIF ptrCommCtrl^.sCmd = 'FBST' THEN
		// Get the DEVice ID
		stat.sPositionControlStatus	:= parsed_reply;
		M_GetPositionControlStatus(s_Test_String);
	ELSIF ptrCommCtrl^.sCmd = 'MLS 4 1' THEN
		// Get Calibration Values
		stat.sCalibrationValues	:= parsed_reply;
		M_GetCalibrationValues(parsed_reply, 1);
	ELSIF ptrCommCtrl^.sCmd = 'MLS 4 2' THEN
		// Get Calibration Values
		stat.sCalibrationValues	:= parsed_reply;
		M_GetCalibrationValues(parsed_reply, 2);
	ELSIF ptrCommCtrl^.sCmd = 'MLS 4 3' THEN
		// Get Calibration Values
		stat.sCalibrationValues	:= parsed_reply;
		M_GetCalibrationValues(parsed_reply, 3);
	ELSIF ptrCommCtrl^.sCmd = 'CGVA 4' THEN
		// Get Calibration Values
		stat.sCounterValues	:= parsed_reply;
		M_GetCounterValues(s_Test_Calibrstion_string);
	ELSIF FIND(ptrCommCtrl^.sCmd,'FBEN') > 0 THEN
		// Enable Servo Drive Mode
		stat.sServoDriveStatus := parsed_reply;
		IF FIND(parsed_reply,'enabled') > 0 THEN
			stat.bServoDrive := TRUE;
		END_IF
	ELSIF ptrCommCtrl^.sCmd = 'FBXT' THEN
		// Disable Servo Drive Mode
		stat.sServoDriveStatus := parsed_reply;
		IF FIND(parsed_reply,'disabled') > 0 THEN
			stat.bServoDrive := FALSE;
		END_IF	
	
		
	END_IF
	M_ReadReply	:= TRUE; (* OK *)
ELSE
	M_ReadReply	:= FALSE;	//	Failed to read from the reply
END_IF
END_METHOD

METHOD M_SetChanState
VAR_INPUT
	nStatus:	UDINT;	// Channel Status as UINT (WORD)
END_VAR
(*
// Get Channel State as a number.
stat.nCH_STATE	:= nStatus;

//
// Extract Channel state from the status word.
//
stat.stState.bACTIVELY_MOVING			:= UDINT_TO_BOOL(nStatus AND E_SA_CH_STATE.BIT_ACTIVELY_MOVING);
stat.stState.bCLOSED_LOOP_ACTIVE		:= UDINT_TO_BOOL(nStatus AND E_SA_CH_STATE.BIT_CLOSED_LOOP_ACTIVE);
stat.stState.bCALIBRATING				:= UDINT_TO_BOOL(nStatus AND E_SA_CH_STATE.BIT_CALIBRATING);
stat.stState.bREFERENCING				:= UDINT_TO_BOOL(nStatus AND E_SA_CH_STATE.BIT_REFERENCING);
stat.stState.bMOVE_DELAYED				:= UDINT_TO_BOOL(nStatus AND E_SA_CH_STATE.BIT_MOVE_DELAYED);
stat.stState.bSENSOR_PRESENT			:= UDINT_TO_BOOL(nStatus AND E_SA_CH_STATE.BIT_SENSOR_PRESENT);
stat.stState.bIS_CALIBRATED				:= UDINT_TO_BOOL(nStatus AND E_SA_CH_STATE.BIT_IS_CALIBRATED);
stat.stState.bIS_REFERENCED				:= UDINT_TO_BOOL(nStatus AND E_SA_CH_STATE.BIT_IS_REFERENCED);
stat.stState.bEND_STOP_REACHED			:= UDINT_TO_BOOL(nStatus AND E_SA_CH_STATE.BIT_END_STOP_REACHED);
stat.stState.bRANGE_LIMIT_REACHED		:= UDINT_TO_BOOL(nStatus AND E_SA_CH_STATE.BIT_RANGE_LIMIT_REACHED);
stat.stState.bFOLLOWING_LIMIT_REACHED	:= UDINT_TO_BOOL(nStatus AND E_SA_CH_STATE.BIT_FOLLOWING_LIMIT_REACHED);
stat.stState.bMOVEMENT_FAILED			:= UDINT_TO_BOOL(nStatus AND E_SA_CH_STATE.BIT_MOVEMENT_FAILED);
stat.stState.bIS_STREAMING				:= UDINT_TO_BOOL(nStatus AND E_SA_CH_STATE.BIT_IS_STREAMING);
stat.stState.bPOSITIONER_OVERLOAD		:= UDINT_TO_BOOL(nStatus AND E_SA_CH_STATE.BIT_POSITIONER_OVERLOAD);
stat.stState.bOVER_TEMPERATURE			:= UDINT_TO_BOOL(nStatus AND E_SA_CH_STATE.BIT_OVER_TEMPERATURE);
stat.stState.bREFERENCE_MARK			:= UDINT_TO_BOOL(nStatus AND E_SA_CH_STATE.BIT_REFERENCE_MARK);
stat.stState.bIS_PHASED					:= UDINT_TO_BOOL(nStatus AND E_SA_CH_STATE.BIT_IS_PHASED);
stat.stState.bPOSITIONER_FAULT			:= UDINT_TO_BOOL(nStatus AND E_SA_CH_STATE.BIT_POSITIONER_FAULT);
stat.stState.bAMPLIFIER_ENABLED			:= UDINT_TO_BOOL(nStatus AND E_SA_CH_STATE.BIT_AMPLIFIER_ENABLED);
stat.stState.bIN_POSITION				:= UDINT_TO_BOOL(nStatus AND E_SA_CH_STATE.BIT_IN_POSITION);


IF	stat.stState.bRANGE_LIMIT_REACHED		OR
	stat.stState.bEND_STOP_REACHED			OR
	stat.stState.bFOLLOWING_LIMIT_REACHED	OR
	stat.stState.bMOVEMENT_FAILED			OR
	stat.stState.bPOSITIONER_OVERLOAD		OR
	stat.stState.bOVER_TEMPERATURE			OR
	stat.stState.bPOSITIONER_FAULT			THEN
		stat.stState.bERROR	:= TRUE;
		stat.bError			:= TRUE;
		stat.sErrorText		:= 'Positioner failure';
		stat.nPosState 		:= E_SA_POS_SM_STATE.ERROR;
ELSE
	// There is no positioner error but maybe the 
	// communication with the MCS2 controller is lost.
	stat.stState.bERROR	:= FALSE;
	
	// Check errors from the MCS2 controller.
	IF stat.bCtrlCommProblem  OR  stat.nCtrlErrorCode <> 0	THEN
		stat.bError	:= TRUE;
	ELSE
		stat.bError		:= FALSE;
		stat.nErrorCode	:= E_SA_CH_ERROR.OK;
		stat.sErrorText	:= 'OK';
	END_IF
END_IF

*)
END_METHOD

METHOD M_SetCmdList
VAR_INPUT
	//index:			UINT := 0;	// Channel index
END_VAR
VAR
	//nChState:	E_SA_POS_SM_STATE := ptrCH[index]^.stat.nPosState;
	//nChState:	E_SA_POS_SM_STATE := E_SA_POS_SM_STATE.CALIB;
	i:			INT;
	cmd:		STRING;
END_VAR
//
// Copy corresponding list of commands to the list in the 'ctrl' structure.
// The generic list contains # characters !
// Examples: ':MOD#:STAT?', ':CHAN#:POS:TARG?', etc.
// They have to be replaced with Channel or Module number.
//
//CASE nChState OF
CASE stat.nPosState	OF
	
	E_SA_POS_SM_STATE.NOT_READY:
		ctrl.cmdList	:= cfg.cmdList_NOT_READY;
	
	(*E_SA_POS_SM_STATE.CALIB:
		// Calibration requires only one command, ':CAL#'.
		ctrl.cmdList[0].cmd			:= 'GFS 1';
		ctrl.cmdList[0].nReplies	:= 1;
		ctrl.cmdList[1].cmd			:= '';		// Command terminator
	*)
	E_SA_POS_SM_STATE.INIT:
		ctrl.cmdList	:= cfg.cmdList_CfgSet;
	
	(*E_SA_POS_SM_STATE.POST_INIT:
		ctrl.cmdList	:= cfg.cmdList_POST_INIT;
	
	E_SA_POS_SM_STATE.CALIB_REF:
		// First set the MIN and MAX limits.
		// Calibrate the REFerence mark. 
		// Read new MIN and MAX limits.
		
		ctrl.cmdList[1].cmd			:= '';
		ctrl.cmdList[1].nReplies	:= 0;
		ctrl.cmdList[2].cmd			:= ':CHAN#:POS ***';
		ctrl.cmdList[2].nReplies	:= 0;
		ctrl.cmdList[3].cmd			:= ':CHAN#:RLIM:MIN?';
		ctrl.cmdList[3].nReplies	:= 1;
		ctrl.cmdList[4].cmd			:= ':CHAN#:RLIM:MAX?';
		ctrl.cmdList[4].nReplies	:= 1;
		ctrl.cmdList[5].cmd			:= '';		// Command terminator
	*)
	E_SA_POS_SM_STATE.READY:
		ctrl.cmdList	:= cfg.cmdList_Mon;
	
	E_SA_POS_SM_STATE.OP:
		ctrl.cmdList	:= cfg.cmdList_Mon;
		//ctrl.cmdList	:= cfg.cmdList_enable_servo_drive;
		
	
	
	E_SA_POS_SM_STATE.BASE_DRIVE_MODE: // Janssen controller Basic Drive Mode 
	
	E_SA_POS_SM_STATE.MOVING:
		// Move the positioner. 
		// Set direction ':CHAN#:VEL <vel>'
		// Set velocity ':CHAN#:VEL <vel>'
		// Move         ':MOVE# <pos>'.
		
		//Command MOV [ADDR] [DIR] [FREQ] [RSS] [STEPS] [TEMP] [STAGE] [DF]
		//Command (example) MOV 1 1 600 100 0 293 CLA2601 1
		//Response (example) Actuating the stage.

		ctrl.cmdList[0].cmd			:= 'MOV 1 1 600 100 0 293 CLA2601 1';
		ctrl.cmdList[0].nReplies	:= 1;
		ctrl.cmdList[1].cmd			:= '';
		ctrl.cmdList[1].nReplies	:= 0;
		//ctrl.cmdList[0].cmd			:= ':CHAN#:VEL ***';
		//ctrl.cmdList[0].nReplies	:= 0;
		//ctrl.cmdList[1].cmd			:= ':MOVE# ***';
		//ctrl.cmdList[1].nReplies	:= 0;
		//ctrl.cmdList[2].cmd			:= '';		// Command terminator
	
	E_SA_POS_SM_STATE.STOP:
		// Stop the positioner. 
		// Requires only one command, ':STOP#'.
		//Command STP [ADDR]
		//Command (example) STP 1
		//Response (example) Stopping the stage.
		
		ctrl.cmdList[0].cmd			:= 'STP 3';
		ctrl.cmdList[0].nReplies	:= 1;
		ctrl.cmdList[1].cmd			:= '';
		ctrl.cmdList[0].nReplies	:= 0;		// Command terminator
	
	E_SA_POS_SM_STATE.FLEX_DRIVE_MODE: // Janssen controller external input mode
		ctrl.cmdList	:= cfg.cmdList_enable_flex_drive;
	
	E_SA_POS_SM_STATE.SERVO_DRIVE_MODE: // Janssen controller Servo Drive Mode
		ctrl.cmdList	:= cfg.cmdList_enable_servo_drive;
		
	E_SA_POS_SM_STATE.DISABLE_SERVO_DRIVE_MODE: // Janssen controller Servo Drive Mode
		ctrl.cmdList	:= cfg.cmdList_disable_servo_drive;
		

	E_SA_POS_SM_STATE.MOVING_TO_SETPOINT:// 3 positioners are Moving to their respective set points in Servo Drive Mode
		ctrl.cmdList	:= cfg.cmdList_moving_to_setpoint;

	E_SA_POS_SM_STATE.EMERGENCY_STOP:    // Emergency stop to halt the positioners
		ctrl.cmdList	:= cfg.cmdList_emergency_stop;
	


	E_SA_POS_SM_STATE.ERROR:
		ctrl.cmdList	:= cfg.cmdList_Mon;
END_CASE

(*
// Set MOD or CHAN index, depending on the command.
FOR i:=0 TO 15 DO
	cmd	:= ctrl.cmdList[i].cmd;
	IF cmd <> ''	THEN
		IF FIND(cmd, ':MOD#') = 1	THEN
			// A MODule command. Set MOD index.
			ctrl.cmdList[i].cmd			:= ptrCH[index]^.M_SetCommandModule(cmd);
		ELSIF FIND(cmd, ':CHAN#') = 1  OR  FIND(cmd, ':MOVE#') = 1	THEN
			// Channel commands.
			// Commands with parameters have the dummy string '***'.
			// Replace *** in generic command with the value.
			IF FIND(cmd, '***') > 0 THEN
				cmd	:= ptrCH[index]^.M_SetCommandValue(cmd);
			END_IF
			// Set CHAN number in the command.
			ctrl.cmdList[i].cmd			:= ptrCH[index]^.M_SetCommandChannel(cmd);
		ELSIF FIND(cmd, ':CAL#') = 1  OR  FIND(cmd, ':REF#') = 1  OR  FIND(cmd, ':STOP#') = 1	THEN
			// Channel command. Replace only the channel number.
			ctrl.cmdList[i].cmd			:= ptrCH[index]^.M_SetCommandChannel(cmd);
		END_IF
	END_IF
END_FOR
*)
END_METHOD

//
// Set next positioner State Machine State.
// This is done at the end of command list execution.
// It Returns TRUE if the state has changed.
//
METHOD M_SetNextPosState : BOOL
VAR_INPUT
END_VAR
CASE stat.nPosState OF
	
	
	E_SA_POS_SM_STATE.NOT_READY:
		IF ch_ctrl.nCmd = E_SA_CH_CMD.REF	THEN
			ch_ctrl.nCmd 			:= E_SA_CH_CMD.NONE;	// Reset command
			stat.nPosState 		:= E_SA_POS_SM_STATE.INIT;
			stat.sStatus		:= 'Referencing/INIT Started';
			M_SetState(E_SA_POS_ELT_STATE.NOTOP);
			M_SetSubstate(E_SA_POS_ELT_SUBSTATE.NOTOP_INITIALIZING);
			M_SetNextPosState	:= TRUE;	// State HAS changed
			
			stat.sRandomtext_1 := 'State from NOT Ready TO INIT';
		ELSE
			M_SetNextPosState	:= FALSE;	// State has NOT changed
		END_IF	
		
		
				
	E_SA_POS_SM_STATE.INIT:
		ch_ctrl.nCmd 			:= E_SA_CH_CMD.NONE;	// Reset command
		stat.nPosState 		:= E_SA_POS_SM_STATE.READY;
		stat.bInitialised	:= TRUE;
		stat.sStatus		:= 'Reference mark calibrated - initialised';
		M_SetState(E_SA_POS_ELT_STATE.NOTOP);
        M_SetSubstate(E_SA_POS_ELT_SUBSTATE.NOTOP_READY);
		M_SetNextPosState	:= TRUE;	// State HAS changed
		
		stat.sRandomtext_2 := 'State from INIT TO READY';


	E_SA_POS_SM_STATE.READY:
		IF ch_ctrl.nCmd = E_SA_CH_CMD.ENABLE	THEN
			ch_ctrl.nCmd 			:= E_SA_CH_CMD.NONE;	// Reset command
			stat.nPosState 		:= E_SA_POS_SM_STATE.SERVO_DRIVE_MODE;
			M_SetNextPosState	:= TRUE;	// State HAS changed
			
			stat.sRandomtext_3 := 'State from READY TO SERVO_DRIVE_MODE';
			
		ELSIF ch_ctrl.nCmd = E_SA_CH_CMD.RESET	THEN			
			ch_ctrl.nCmd 			:= E_SA_CH_CMD.NONE;	// Reset command
			stat.nPosState 		:= E_SA_POS_SM_STATE.NOT_READY;
			stat.bInitialised	:= FALSE;
			stat.nErrorCode		:= E_SM_ERROR.OK; 
			stat.sErrorText		:= 'OK';
			stat.sStatus		:= 'Positioner Reset';
			M_SetState(E_SA_POS_ELT_STATE.NOTOP);
			M_SetSubstate(E_SA_POS_ELT_SUBSTATE.NOTOP_NOTREADY);
			M_SetNextPosState	:= TRUE;	// State HAS changed
		
		ELSE
			M_SetNextPosState	:= FALSE;	// State has NOT changed
		END_IF

	E_SA_POS_SM_STATE.SERVO_DRIVE_MODE:
		ch_ctrl.nCmd 			:= E_SA_CH_CMD.NONE;	// Reset command
		stat.nPosState 		:= E_SA_POS_SM_STATE.OP;
		//stat.sStatus		:= 'Operational';
		//M_SetState(E_SA_POS_ELT_STATE.OP);
		//M_SetSubstate(E_SA_POS_ELT_SUBSTATE.OP_STANDSTILL);
		M_SetNextPosState	:= TRUE;	// State HAS changed
		
		stat.sRandomtext_4 := 'State from READY To OP' ;	
	
	E_SA_POS_SM_STATE.OP:
		IF	ch_ctrl.nCmd = E_SA_CH_CMD.MOV THEN
			ch_ctrl.nCmd 			:= E_SA_CH_CMD.NONE;	// Reset command
			stat.nPosState 		:= E_SA_POS_SM_STATE.MOVING_TO_SETPOINT;
			stat.stState.bACTIVELY_MOVING	:= TRUE;
			stat.stState.bIN_POSITION		:= FALSE;
			//stat.nLastPosState 	:= E_SA_POS_SM_STATE.OP;
			//stat.sStatus		:= 'Moving to a setpoint...';
			//M_SetSubstate(E_SA_POS_ELT_SUBSTATE.OP_MOVING);	
			M_SetNextPosState	:= TRUE;	// State HAS changed
			
			stat.sRandomtext_5 := 'State from OP TO MOVING_TO_SETPOINT';
		
		ELSIF ch_ctrl.nCmd = E_SA_CH_CMD.DISABLE	THEN
			ch_ctrl.nCmd 		:= E_SA_CH_CMD.NONE;	// Reset command
			stat.nPosState 		:= E_SA_POS_SM_STATE.DISABLE_SERVO_DRIVE_MODE;
			M_SetNextPosState	:= TRUE;	// State HAS changed
			
		ELSIF ch_ctrl.nCmd = E_SA_CH_CMD.RESET	THEN			
			ch_ctrl.nCmd 		:= E_SA_CH_CMD.NONE;	// Reset command
			stat.nPosState 		:= E_SA_POS_SM_STATE.NOT_READY;
			stat.bInitialised	:= FALSE;
			stat.nErrorCode		:= E_SM_ERROR.OK; 
			stat.sErrorText		:= 'OK';
			stat.sStatus		:= 'Positioner Reset';
			M_SetState(E_SA_POS_ELT_STATE.NOTOP);
			M_SetSubstate(E_SA_POS_ELT_SUBSTATE.NOTOP_NOTREADY);
			M_SetNextPosState	:= TRUE;	// State HAS changed
		
		ELSE
			M_SetNextPosState	:= FALSE;	// State has NOT changed
		END_IF
	
	E_SA_POS_SM_STATE.DISABLE_SERVO_DRIVE_MODE:
		ch_ctrl.nCmd 			:= E_SA_CH_CMD.NONE;	// Reset command
		stat.nPosState 		:= E_SA_POS_SM_STATE.READY;
		//stat.sStatus		:= 'Ready';
		//M_SetState(E_SA_POS_ELT_STATE.NOTOP);
		//M_SetSubstate(E_SA_POS_ELT_SUBSTATE.NOTOP_READY);
		M_SetNextPosState	:= TRUE;	// State HAS changed
		
		stat.sRandomtext_6 := 'DISABLE_SERVO_DRIVE To Ready' ;
	
	
	E_SA_POS_SM_STATE.MOVING_TO_SETPOINT:
		IF ch_ctrl.nCmd = E_SA_CH_CMD.STOP THEN
			ch_ctrl.nCmd 			:= E_SA_CH_CMD.NONE;	// Reset command
			stat.nPosState 		:= E_SA_POS_SM_STATE.EMERGENCY_STOP;			
			//stat.sStatus		:= 'Stopping...';
			//M_SetSubstate(E_SA_POS_ELT_SUBSTATE.OP_STOPPING);
			M_SetNextPosState	:= TRUE;	// State HAS changed
			
			stat.sRandomtext_7 := 'State from MOVING_TO_SET_POINT To EMERGENCY_STOP' ;
		ELSE
			stat.nPosState := E_SA_POS_SM_STATE.OP;
			M_SetNextPosState	:= TRUE;	// State HAS changed
		END_IF
		
	E_SA_POS_SM_STATE.EMERGENCY_STOP:
		stat.nPosState := E_SA_POS_SM_STATE.OP;
		stat.sStatus		:= 'Positioner Stopped';
		M_SetNextPosState	:= TRUE;	// State HAS changed

	E_SA_POS_SM_STATE.ERROR:
		IF ch_ctrl.nCmd = E_SA_CH_CMD.REF	THEN
			ch_ctrl.nCmd 			:= E_SA_CH_CMD.NONE;	// Reset command
			stat.nPosState 		:= E_SA_POS_SM_STATE.INIT;
			stat.bInitialised	:= FALSE;
			stat.sStatus		:= 'Referencing/INIT Started';
			M_SetState(E_SA_POS_ELT_STATE.NOTOP);
			M_SetSubstate(E_SA_POS_ELT_SUBSTATE.NOTOP_NOTREADY);
			M_SetNextPosState	:= TRUE;	// State HAS changed
			
		ELSE
			stat.sStatus		:= M_GetErrorString();
			M_SetNextPosState	:= FALSE;	// State has NOT changed
		END_IF
		
END_CASE




(*

CASE stat.nPosState OF
	
	
	E_SA_POS_SM_STATE.NOT_READY:
				
		//IF ch_ctrl.nCmd = E_SA_CH_CMD.REF	THEN
			ch_ctrl.nCmd 			:= E_SA_CH_CMD.NONE;	// Reset command
			stat.nPosState 		:= E_SA_POS_SM_STATE.INIT;
			stat.sStatus		:= 'Referencing/INIT Started';
			M_SetState(E_SA_POS_ELT_STATE.NOTOP);
			M_SetSubstate(E_SA_POS_ELT_SUBSTATE.NOTOP_INITIALIZING);
			M_SetNextPosState	:= TRUE;	// State HAS changed
			
			stat.sRandomtext_1 := 'Not Ready done';
		//ELSE
		//	M_SetNextPosState	:= FALSE;	// State has NOT changed
		//END_IF
		
	// Janssen
	E_SA_POS_SM_STATE.INIT:
		stat.nPosState 	:= E_SA_POS_SM_STATE.READY;	// was READY
		stat.nLastPosState := E_SA_POS_SM_STATE.INIT;
		stat.bInitialised	:= TRUE;
		stat.sStatus		:= 'Reference mark calibrated - initialised';
		M_SetState(E_SA_POS_ELT_STATE.NOTOP);
        M_SetSubstate(E_SA_POS_ELT_SUBSTATE.NOTOP_READY);
		M_SetNextPosState	:= TRUE;	// State HAS changed
		
		stat.sRandomtext_2 := 'INIT done';

	E_SA_POS_SM_STATE.READY:
		stat.sRandomtext_3 := 'In Ready';
		IF ch_ctrl.nCmd = E_SA_CH_CMD.ENABLE	THEN
		
			ch_ctrl.nCmd 			:= E_SA_CH_CMD.NONE;	// Reset command
			stat.nPosState 		:= E_SA_POS_SM_STATE.SERVO_DRIVE_MODE;
			stat.nLastPosState := E_SA_POS_SM_STATE.READY;
			stat.sStatus		:= 'Operational';
			M_SetState(E_SA_POS_ELT_STATE.OP);
			M_SetSubstate(E_SA_POS_ELT_SUBSTATE.OP_STANDSTILL);
			M_SetNextPosState	:= TRUE;	// State HAS changed
			
			stat.sRandomtext_4 := 'Executed Enable done';
		
		ELSIF ch_ctrl.nCmd = E_SA_CH_CMD.RESET	THEN
		
			stat.sRandomtext_5 := 'inside RESET';
			
			ch_ctrl.nCmd 			:= E_SA_CH_CMD.NONE;	// Reset command
			stat.nPosState 		:= E_SA_POS_SM_STATE.NOT_READY;
			stat.bInitialised	:= FALSE;
			//stat.nErrorCode		:= E_SA_CH_ERROR.OK; 
			stat.nErrorCode		:= E_SM_ERROR.OK; 
			stat.sErrorText		:= 'OK';
			stat.sStatus		:= 'Positioner Reset';
			M_SetState(E_SA_POS_ELT_STATE.NOTOP);
			M_SetSubstate(E_SA_POS_ELT_SUBSTATE.NOTOP_NOTREADY);
			M_SetNextPosState	:= TRUE;	// State HAS changed
			
			
		ELSE
			M_SetNextPosState	:= FALSE;	// State has NOT changed
		END_IF
		
	
	E_SA_POS_SM_STATE.OP:
		
		stat.sRandomtext_6 := 'Inside OP state';
		
		IF ch_ctrl.nCmd = E_SA_CH_CMD.RESET	THEN
			ch_ctrl.nCmd 			:= E_SA_CH_CMD.NONE;	// Reset command
			stat.nPosState 		:= E_SA_POS_SM_STATE.NOT_READY;
			stat.bInitialised	:= FALSE;
			//stat.nErrorCode		:= E_SA_CH_ERROR.OK; 
			stat.nErrorCode		:= E_SM_ERROR.OK;
			stat.sErrorText		:= 'OK';
			stat.sStatus		:= 'Positioner Reset';
			M_SetState(E_SA_POS_ELT_STATE.NOTOP);
			M_SetSubstate(E_SA_POS_ELT_SUBSTATE.NOTOP_NOTREADY);
			M_SetNextPosState	:= TRUE;	// State HAS changed
		ELSIF ch_ctrl.nCmd = E_SA_CH_CMD.DISABLE	THEN
			ch_ctrl.nCmd 			:= E_SA_CH_CMD.NONE;	// Reset command
			stat.nPosState 		:= E_SA_POS_SM_STATE.READY;
			stat.sStatus		:= 'Ready';
			M_SetState(E_SA_POS_ELT_STATE.NOTOP);
			M_SetSubstate(E_SA_POS_ELT_SUBSTATE.NOTOP_READY);
			M_SetNextPosState	:= TRUE;	// State HAS changed
			
			stat.sRandomtext_7 := 'DISABLE executed';
			
		ELSIF ch_ctrl.nCmd = E_SA_CH_CMD.MOVE_TO_SETPOINT	THEN
			ch_ctrl.nCmd 			:= E_SA_CH_CMD.NONE;	// Reset command
			stat.stState.bACTIVELY_MOVING	:= TRUE;
			stat.stState.bIN_POSITION		:= FALSE;
			stat.nPosState 		:= E_SA_POS_SM_STATE.MOVING_TO_SETPOINT;
			stat.nLastPosState 	:= E_SA_POS_SM_STATE.OP;
			stat.sStatus		:= 'Moving to a setpoint...';
			M_SetSubstate(E_SA_POS_ELT_SUBSTATE.OP_MOVING);
			M_SetNextPosState	:= TRUE;	// State HAS changed
		ELSIF ch_ctrl.nCmd = E_SA_CH_CMD.EMERGENCY_STOP	THEN
			ch_ctrl.nCmd 			:= E_SA_CH_CMD.NONE;	// Reset command
			stat.nPosState 		:= E_SA_POS_SM_STATE.STOP;
			stat.sStatus		:= 'Stopping...';
			M_SetSubstate(E_SA_POS_ELT_SUBSTATE.OP_STOPPING);
			M_SetNextPosState	:= TRUE;	// State HAS changed
		ELSIF	NOT stat.stState.bACTIVELY_MOVING	AND
				// check this
				stat.stState.bIN_POSITION			AND
				stat.nLastPosState <> E_SA_POS_SM_STATE.CALIB_REF	THEN
					stat.sStatus		:= 'Move completed';
					M_SetNextPosState	:= FALSE;	// State has NOT changed	
		ELSIF ch_ctrl.nCmd = E_SA_CH_CMD.DISABLE_SERVO_DRIVE	THEN
			ch_ctrl.nCmd 			:= E_SA_CH_CMD.NONE;	// Reset command
			stat.nPosState 		:= E_SA_POS_SM_STATE.OP;
			stat.sStatus		:= 'Operational';
			M_SetState(E_SA_POS_ELT_STATE.OP);
			M_SetSubstate(E_SA_POS_ELT_SUBSTATE.OP_STANDSTILL);
			M_SetNextPosState	:= TRUE;	// State HAS changed
		ELSIF ch_ctrl.nCmd = E_SA_CH_CMD.RESET	THEN
			ch_ctrl.nCmd 			:= E_SA_CH_CMD.NONE;	// Reset command
			stat.nPosState 		:= E_SA_POS_SM_STATE.NOT_READY;
			stat.bInitialised	:= FALSE;
			//stat.nErrorCode		:= E_SA_CH_ERROR.OK; 
			stat.nErrorCode		:= E_SM_ERROR.OK;
			stat.sErrorText		:= 'OK';
			stat.sStatus		:= 'Positioner Reset';
			M_SetState(E_SA_POS_ELT_STATE.NOTOP);
			M_SetSubstate(E_SA_POS_ELT_SUBSTATE.NOTOP_NOTREADY);
			M_SetNextPosState	:= TRUE;	// State HAS changed
		
		ELSE
			M_SetNextPosState	:= FALSE;	// State has NOT changed
		END_IF
		
		stat.sRandomtext_7 := 'Exiting OP state';
	(*	
	// Basic Drive Mode
	E_SA_POS_SM_STATE.BASE_DRIVE_MODE:
		IF ch_ctrl.nCmd = E_SA_CH_CMD.MOV	THEN
			ch_ctrl.nCmd 			:= E_SA_CH_CMD.NONE;	// Reset command
			stat.stState.bACTIVELY_MOVING	:= TRUE;
			stat.stState.bIN_POSITION		:= FALSE;
			stat.nPosState 		:= E_SA_POS_SM_STATE.MOVING;
			stat.nLastPosState 	:= E_SA_POS_SM_STATE.OP;
			stat.sStatus		:= 'Moving...';
			M_SetSubstate(E_SA_POS_ELT_SUBSTATE.OP_MOVING);
			M_SetNextPosState	:= TRUE;	// State HAS changed
		ELSIF ch_ctrl.nCmd = E_SA_CH_CMD.STOP	THEN
			ch_ctrl.nCmd 			:= E_SA_CH_CMD.NONE;	// Reset command
			stat.nPosState 		:= E_SA_POS_SM_STATE.STOP;
			stat.sStatus		:= 'Stopping...';
			M_SetSubstate(E_SA_POS_ELT_SUBSTATE.OP_STOPPING);
			M_SetNextPosState	:= TRUE;	// State HAS changed
		ELSIF	NOT stat.stState.bACTIVELY_MOVING	AND
				// Check this and Servo drive mode
				stat.stState.bIN_POSITION			AND
				stat.nLastPosState <> E_SA_POS_SM_STATE.CALIB_REF	THEN
					stat.sStatus		:= 'Move completed';
					M_SetNextPosState	:= FALSE;	// State has NOT changed	
		ELSIF ch_ctrl.nCmd = E_SA_CH_CMD.DISABLE_BASE_DRIVE	THEN
			ch_ctrl.nCmd 			:= E_SA_CH_CMD.NONE;	// Reset command
			stat.nPosState 		:= E_SA_POS_SM_STATE.OP;
			stat.sStatus		:= 'Operational';
			M_SetState(E_SA_POS_ELT_STATE.OP);
			M_SetSubstate(E_SA_POS_ELT_SUBSTATE.OP_STANDSTILL);
			M_SetNextPosState	:= TRUE;	// State HAS changed
		ELSIF ch_ctrl.nCmd = E_SA_CH_CMD.RESET	THEN
			ch_ctrl.nCmd 			:= E_SA_CH_CMD.NONE;	// Reset command
			stat.nPosState 		:= E_SA_POS_SM_STATE.NOT_READY;
			stat.bInitialised	:= FALSE;
			//stat.nErrorCode		:= E_SA_CH_ERROR.OK; 
			stat.nErrorCode		:= E_SM_ERROR.OK;
			stat.sErrorText		:= 'OK';
			stat.sStatus		:= 'Positioner Reset';
			M_SetState(E_SA_POS_ELT_STATE.NOTOP);
			M_SetSubstate(E_SA_POS_ELT_SUBSTATE.NOTOP_NOTREADY);
			M_SetNextPosState	:= TRUE;	// State HAS changed
		ELSE
			M_SetNextPosState	:= FALSE;	// State has NOT changed	
		END_IF
	
	E_SA_POS_SM_STATE.MOVING:
		IF ch_ctrl.nCmd = E_SA_CH_CMD.STOP	THEN
			ch_ctrl.nCmd 			:= E_SA_CH_CMD.NONE;	// Reset command
			stat.nPosState 		:= E_SA_POS_SM_STATE.STOP;
			stat.sStatus		:= 'Stopping...';
			M_SetSubstate(E_SA_POS_ELT_SUBSTATE.OP_STOPPING);
			M_SetNextPosState	:= TRUE;	// State HAS changed
		ELSE
			stat.nPosState := E_SA_POS_SM_STATE.OP;
			M_SetNextPosState	:= TRUE;	// State HAS changed
		END_IF
	
	E_SA_POS_SM_STATE.STOP:
		stat.nPosState := E_SA_POS_SM_STATE.BASE_DRIVE_MODE;
		stat.sStatus		:= 'Positioner Stopped';
		M_SetNextPosState	:= TRUE;	// State HAS changed
	
	// Flex Drive Mode (External Input)
	E_SA_POS_SM_STATE.FLEX_DRIVE_MODE:
		IF  ch_ctrl.nCmd = E_SA_CH_CMD.DISABLE_FLEX_DRIVE	THEN
			ch_ctrl.nCmd 			:= E_SA_CH_CMD.NONE;	// Reset command
			stat.nPosState 		:= E_SA_POS_SM_STATE.OP;
			stat.sStatus		:= 'Operational';
			M_SetState(E_SA_POS_ELT_STATE.OP);
			M_SetSubstate(E_SA_POS_ELT_SUBSTATE.OP_STANDSTILL);
			M_SetNextPosState	:= TRUE;	// State HAS changed
		ELSE
			M_SetNextPosState	:= FALSE;	// State has NOT changed	
		END_IF
	*)
	
	// Servo Drive Mode
	E_SA_POS_SM_STATE.SERVO_DRIVE_MODE:
		stat.sRandomtext_6 := 'Inside Servodrive Mode';
		IF ch_ctrl.nCmd = E_SA_CH_CMD.MOVE_TO_SETPOINT	THEN
			ch_ctrl.nCmd 			:= E_SA_CH_CMD.NONE;	// Reset command
			stat.stState.bACTIVELY_MOVING	:= TRUE;
			stat.stState.bIN_POSITION		:= FALSE;
			stat.nPosState 		:= E_SA_POS_SM_STATE.MOVING_TO_SETPOINT;
			stat.nLastPosState 	:= E_SA_POS_SM_STATE.OP;
			stat.sStatus		:= 'Moving to a setpoint...';
			M_SetSubstate(E_SA_POS_ELT_SUBSTATE.OP_MOVING);
			M_SetNextPosState	:= TRUE;	// State HAS changed
		ELSIF ch_ctrl.nCmd = E_SA_CH_CMD.EMERGENCY_STOP	THEN
			ch_ctrl.nCmd 			:= E_SA_CH_CMD.NONE;	// Reset command
			stat.nPosState 		:= E_SA_POS_SM_STATE.STOP;
			stat.sStatus		:= 'Stopping...';
			M_SetSubstate(E_SA_POS_ELT_SUBSTATE.OP_STOPPING);
			M_SetNextPosState	:= TRUE;	// State HAS changed
		ELSIF	NOT stat.stState.bACTIVELY_MOVING	AND
				// check this
				stat.stState.bIN_POSITION			AND
				stat.nLastPosState <> E_SA_POS_SM_STATE.CALIB_REF	THEN
					stat.sStatus		:= 'Move completed';
					M_SetNextPosState	:= FALSE;	// State has NOT changed	
		ELSIF ch_ctrl.nCmd = E_SA_CH_CMD.DISABLE_SERVO_DRIVE	THEN
			ch_ctrl.nCmd 			:= E_SA_CH_CMD.NONE;	// Reset command
			stat.nPosState 		:= E_SA_POS_SM_STATE.OP;
			stat.sStatus		:= 'Operational';
			M_SetState(E_SA_POS_ELT_STATE.OP);
			M_SetSubstate(E_SA_POS_ELT_SUBSTATE.OP_STANDSTILL);
			M_SetNextPosState	:= TRUE;	// State HAS changed
		ELSIF ch_ctrl.nCmd = E_SA_CH_CMD.RESET	THEN
			ch_ctrl.nCmd 			:= E_SA_CH_CMD.NONE;	// Reset command
			stat.nPosState 		:= E_SA_POS_SM_STATE.NOT_READY;
			stat.bInitialised	:= FALSE;
			//stat.nErrorCode		:= E_SA_CH_ERROR.OK; 
			stat.nErrorCode		:= E_SM_ERROR.OK;
			stat.sErrorText		:= 'OK';
			stat.sStatus		:= 'Positioner Reset';
			M_SetState(E_SA_POS_ELT_STATE.NOTOP);
			M_SetSubstate(E_SA_POS_ELT_SUBSTATE.NOTOP_NOTREADY);
			M_SetNextPosState	:= TRUE;	// State HAS changed
		ELSE
			M_SetNextPosState	:= FALSE;	// State has NOT changed	
		END_IF
		
	
	E_SA_POS_SM_STATE.MOVING_TO_SET_POINT:
		IF ch_ctrl.nCmd = E_SA_CH_CMD.EMERGENCY_STOP	THEN
			ch_ctrl.nCmd 			:= E_SA_CH_CMD.NONE;	// Reset command
			stat.nPosState 		:= E_SA_POS_SM_STATE.STOP;
			stat.sStatus		:= 'Stopping...';
			M_SetSubstate(E_SA_POS_ELT_SUBSTATE.OP_STOPPING);
			M_SetNextPosState	:= TRUE;	// State HAS changed
		ELSIF ch_ctrl.nCmd = E_SA_CH_CMD.SET_POINT_ACHIEVED	THEN
			ch_ctrl.nCmd 			:= E_SA_CH_CMD.NONE;	// Reset command
			stat.stState.bSERVO_DRIVE_ENABLED	:= TRUE;
			//stat.stState.bIN_POSITION		:= FALSE;
			stat.nPosState 		:= E_SA_POS_SM_STATE.SERVO_DRIVE_MODE;
			stat.nLastPosState 	:= E_SA_POS_SM_STATE.OP;
			stat.sStatus		:= 'Servo Drive Enabled';
			M_SetSubstate(E_SA_POS_ELT_SUBSTATE.NOTOP_READY);
			M_SetNextPosState	:= TRUE;	// State HAS changed
		ELSIF	NOT stat.stState.bACTIVELY_MOVING	AND
				// Check this and Servo drive mode
				stat.stState.bIN_POSITION			AND
				stat.nLastPosState <> E_SA_POS_SM_STATE.CALIB_REF	THEN
					stat.sStatus		:= 'Move completed';
					M_SetNextPosState	:= FALSE;	// State has NOT changed
		ELSE
			M_SetNextPosState	:= FALSE;	// State has NOT changed	
		END_IF
	
	E_SA_POS_SM_STATE.EMERGENCY_STOP:
		stat.nPosState := E_SA_POS_SM_STATE.SERVO_DRIVE_MODE;
		stat.sStatus		:= 'Positioner Stopped';
		M_SetNextPosState	:= TRUE;	// State HAS changed	
	
	
	
	
